// NETWORK 29
Ramp_Test_0(
    Enable := VCC_Ramp_Test_On,
    uExt := VCC_Ramp_Test_u_DCV_1,
    u0 := 0,
    uRetr := VCC_Ramp_Test_u_DCV_2,
    t0 := VCC_Test_t0,
    tRampUp := VCC_Ramp_Test_tR,
    tHold_Up := VCC_Ramp_Test_tHold_Up,
    tHold_Down := VCC_Ramp_Test_tHold_Down,
    tRampDown := VCC_Ramp_Test_tR,
    tWait := VCC_Ramp_Test_tWait,
    CyclicTime := UDP_Send.plcTime); // Ramp_Test
VCC_Anti_Dead_Band_v2_0(
    u_DCV_ref := Ramp_Test_0.Valve_Opening_Ref,
    DB_Up := VCC_Cntrl_DB_up,
    DB_Down := VCC_Cntrl_DB_down); // VCC_Anti_Dead_Band_v2
LREAL_TO_REAL(VCC_Anti_Dead_Band_v2_0.u_DCV);

// NETWORK 30
Ramp_Test_1(
    Enable := VCC_Ramp_Test_On,
    uExt := VCC_Ramp_Test_u_DCV_1,
    u0 := 0,
    uRetr := VCC_Ramp_Test_u_DCV_2,
    t0 := VCC_Test_t0,
    tRampUp := VCC_Ramp_Test_tR,
    tHold_Up := VCC_Ramp_Test_tHold_Up,
    tHold_Down := VCC_Ramp_Test_tHold_Down,
    tRampDown := VCC_Ramp_Test_tR,
    tWait := VCC_Ramp_Test_tWait,
    CyclicTime := UDP_Send.plcTime); // Ramp_Test
uRamp := LREAL_TO_REAL(Ramp_Test_1.Valve_Opening_Ref);

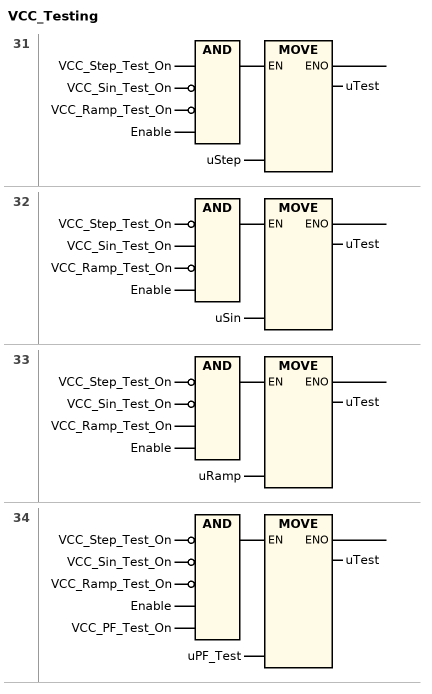
// NETWORK 31
IF VCC_Step_Test_On AND NOT VCC_Sin_Test_On AND NOT VCC_Ramp_Test_On AND Enable THEN uTest := uStep; END_IF

// NETWORK 32
IF NOT VCC_Step_Test_On AND VCC_Sin_Test_On AND NOT VCC_Ramp_Test_On AND Enable THEN uTest := uSin; END_IF

// NETWORK 33
IF NOT VCC_Step_Test_On AND NOT VCC_Sin_Test_On AND VCC_Ramp_Test_On AND Enable THEN uTest := uRamp; END_IF

// NETWORK 34
IF NOT VCC_Step_Test_On AND NOT VCC_Sin_Test_On AND NOT VCC_Ramp_Test_On AND Enable AND VCC_PF_Test_On THEN
    uTest := uPF_Test;
END_IF

END_PROGRAM

// IndraMotionMlc1/Application/VCC_StepFunction_Test
FUNCTION_BLOCK VCC_StepFunction_Test
VAR_INPUT
	Enable: BOOL;
	Extend_Opening_SP: LREAL;
	Neutral_Pos_SP: LREAL;
	Retract_Opening_SP: LREAL;
	CyclicTime: LREAL;
	t0: LREAL;
	t1: LREAL;
	t2: LREAL;
	t3: LREAL;
END_VAR
VAR_OUTPUT
	Valve_Opening_Ref: LREAL;
	EndTime: LREAL;
END_VAR
VAR
	tmp: LREAL;
	temp1: LREAL;
END_VAR


(* MATLAB Function: '<S1>/StepFunction' *)
(* MATLAB Function 'VCC_StepFunction_Test/StepFunction': '<S2>:1' *)
(* '<S2>:1:3' y = Neutral_Pos_SP; *)
(* '<S2>:1:5' if t>=0 &amp;&amp; t<t0 *)

IF (CyclicTime >= 0.0) AND (CyclicTime < t0) THEN 
    (* '<S2>:1:6' y = Neutral_Pos_SP; *)
    Valve_Opening_Ref := Neutral_Pos_SP;
ELSE 
    tmp := t0 + t1;

    IF (CyclicTime >= t0) AND (CyclicTime < tmp) THEN 
        (* '<S2>:1:7' elseif t>=(t0) &amp;&amp; t<(t0+t1) *)
        (* '<S2>:1:8' y = Extend_Opening_SP; *)
        Valve_Opening_Ref := Extend_Opening_SP;
    ELSE 
        temp1 := tmp + t2;

        IF (CyclicTime >= tmp) AND (CyclicTime < temp1) THEN 
            (* '<S2>:1:9' elseif t>=(t0+t1) &amp;&amp; t<(t0+t1+t2) *)
            (* '<S2>:1:10' y = Neutral_Pos_SP; *)
            Valve_Opening_Ref := Neutral_Pos_SP;
        ELSIF (CyclicTime >= temp1) AND (CyclicTime < (temp1 + t3)) THEN 
            (* '<S2>:1:11' elseif t>=(t0+t1+t2) &amp;&amp; t<(t0+t1+t2+t3) *)
            (* '<S2>:1:12' y = Retract_Opening_SP; *)
            Valve_Opening_Ref := Retract_Opening_SP;
        ELSE 
            (* '<S2>:1:13' else *)
            (* '<S2>:1:14' y = Neutral_Pos_SP; *)
            Valve_Opening_Ref := Neutral_Pos_SP;
        END_IF;

    END_IF;

END_IF;

(* Switch: '<S1>/Switch' *)
(* '<S2>:1:17' T = t0+t1+t2+t3; *)

IF  NOT Enable THEN 
    (* Outport: '<Root>/Valve_Opening_Ref' *)
    Valve_Opening_Ref := Neutral_Pos_SP;
END_IF;

(* End of Switch: '<S1>/Switch' *)


(* Outport: '<Root>/EndTime' incorporates:
 *  MATLAB Function: '<S1>/StepFunction' *)
EndTime := ((t0 + t1) + t2) + t3;

END_FUNCTION_BLOCK

// IndraMotionMlc1/Application/PF1
FUNCTION_BLOCK PF1
VAR_INPUT
	ssMethodType: SINT;
	Enable: BOOL;
	usDelay: LREAL;
	kQf: LREAL;
	HPF_Num1: LREAL;
	HPF_Num2: LREAL;
	HPF_Den1: LREAL;
	HPF_Den2: LREAL;
	pAsimbar: LREAL;
	pBsimbar: LREAL;
END_VAR
VAR_OUTPUT
	uPF: LREAL;
END_VAR
VAR
	HP_Filter_tmp: LREAL;
	VectorConcatenate: ARRAY[0..1] OF LREAL;
	VectorConcatenate1: ARRAY[0..1] OF LREAL;
	HP_Filter_states: LREAL;
END_VAR



CASE ssMethodType OF
    0: 
        (* InitializeConditions for DiscreteTransferFcn: '<S1>/HP_Filter' *)
        HP_Filter_states := 0.0;
    1: 
        (* SignalConversion: '<S1>/ConcatBufferAtVector ConcatenateIn1' *)
        VectorConcatenate[0] := HPF_Num1;
        (* SignalConversion: '<S1>/ConcatBufferAtVector ConcatenateIn2' *)
        VectorConcatenate[1] := HPF_Num2;
        (* SignalConversion: '<S1>/ConcatBufferAtVector Concatenate1In1' *)
        VectorConcatenate1[0] := HPF_Den1;
        (* SignalConversion: '<S1>/ConcatBufferAtVector Concatenate1In2' *)
        VectorConcatenate1[1] := HPF_Den2;
        (* DiscreteTransferFcn: '<S1>/HP_Filter' incorporates:
         *  Gain: '<S1>/Gain'
         *  Gain: '<S1>/Gain3'
         *  Gain: '<S1>/muC'
         *  Sum: '<S1>/Add' *)
        HP_Filter_tmp := (((100000.0 * pAsimbar) * 1.4083) - (100000.0 * pBsimbar)) - (VectorConcatenate1[1] * HP_Filter_states);
        (* Switch: '<S1>/Switch2' incorporates:
         *  Constant: '<S1>/Constant' *)

        IF Enable THEN 
            (* Switch: '<S1>/Switch1' incorporates:
             *  Constant: '<S1>/Constant'
             *  DiscreteTransferFcn: '<S1>/HP_Filter'
             *  Product: '<S1>/Product' *)

            IF usDelay > 2.0 THEN 
                uPF := ((VectorConcatenate[0] * HP_Filter_tmp) + (VectorConcatenate[1] * HP_Filter_states)) * kQf;
            ELSE 
                uPF := 0.0;
            END_IF;

            (* End of Switch: '<S1>/Switch1' *)
        ELSE 
            uPF := 0.0;
        END_IF;

        (* End of Switch: '<S1>/Switch2' *)
        

        (* Saturate: '<S1>/Saturation5' *)

        IF uPF >= 1.0 THEN 
            uPF := 1.0;
        ELSIF uPF <= -1.0 THEN 
            uPF := -1.0;
        END_IF;

        (* End of Saturate: '<S1>/Saturation5' *)
        

        (* Update for DiscreteTransferFcn: '<S1>/HP_Filter' *)
        HP_Filter_states := HP_Filter_tmp;
END_CASE;

END_FUNCTION_BLOCK

// IndraMotionMlc1/Application/PF2
FUNCTION_BLOCK PF2
VAR_INPUT
	ssMethodType: SINT;
	Enable: BOOL;
	usDelay: LREAL;
	kQf: LREAL;
	HPF_Num1: LREAL;
	HPF_Num2: LREAL;
	HPF_Den1: LREAL;
	HPF_Den2: LREAL;
	GVI_Num1: LREAL;
	GVI_Num2: LREAL;
	GVI_Num3: LREAL;
	GVI_Den1: LREAL;
	GVI_Den2: LREAL;
	GVI_Den3: LREAL;
	pAsimbar: LREAL;
	pBsimbar: LREAL;
END_VAR
VAR_OUTPUT
	uPF: LREAL;
END_VAR
VAR
	rtb_Add: LREAL;
	HP_Filter_tmp: LREAL;
	VectorConcatenate: ARRAY[0..1] OF LREAL;
	VectorConcatenate1: ARRAY[0..1] OF LREAL;
	VectorConcatenate2: ARRAY[0..2] OF LREAL;
	VectorConcatenate3: ARRAY[0..2] OF LREAL;
	HP_Filter_states: LREAL;
	Gv_Inv_states: ARRAY[0..1] OF LREAL;
END_VAR



CASE ssMethodType OF
    0: 
        (* InitializeConditions for DiscreteTransferFcn: '<S1>/HP_Filter' *)
        HP_Filter_states := 0.0;
        (* InitializeConditions for DiscreteTransferFcn: '<S1>/Gv_Inv' *)
        Gv_Inv_states[0] := 0.0;
        Gv_Inv_states[1] := 0.0;
    1: 
        (* SignalConversion: '<S1>/ConcatBufferAtVector ConcatenateIn1' *)
        VectorConcatenate[0] := HPF_Num1;
        (* SignalConversion: '<S1>/ConcatBufferAtVector ConcatenateIn2' *)
        VectorConcatenate[1] := HPF_Num2;
        (* SignalConversion: '<S1>/ConcatBufferAtVector Concatenate1In1' *)
        VectorConcatenate1[0] := HPF_Den1;
        (* SignalConversion: '<S1>/ConcatBufferAtVector Concatenate1In2' *)
        VectorConcatenate1[1] := HPF_Den2;
        (* DiscreteTransferFcn: '<S1>/HP_Filter' incorporates:
         *  Gain: '<S1>/Gain'
         *  Gain: '<S1>/Gain3'
         *  Gain: '<S1>/muC'
         *  Sum: '<S1>/Add' *)
        HP_Filter_tmp := (((100000.0 * pAsimbar) * 1.4083) - (100000.0 * pBsimbar)) - (VectorConcatenate1[1] * HP_Filter_states);
        (* SignalConversion: '<S1>/ConcatBufferAtVector Concatenate2In1' *)
        VectorConcatenate2[0] := GVI_Num1;
        (* SignalConversion: '<S1>/ConcatBufferAtVector Concatenate2In2' *)
        VectorConcatenate2[1] := GVI_Num2;
        (* SignalConversion: '<S1>/ConcatBufferAtVector Concatenate2In3' *)
        VectorConcatenate2[2] := GVI_Num3;
        (* SignalConversion: '<S1>/ConcatBufferAtVector Concatenate3In1' *)
        VectorConcatenate3[0] := GVI_Den1;
        (* SignalConversion: '<S1>/ConcatBufferAtVector Concatenate3In2' *)
        VectorConcatenate3[1] := GVI_Den2;
        (* SignalConversion: '<S1>/ConcatBufferAtVector Concatenate3In3' *)
        VectorConcatenate3[2] := GVI_Den3;
        (* DiscreteTransferFcn: '<S1>/Gv_Inv' incorporates:
         *  DiscreteTransferFcn: '<S1>/HP_Filter'
         *  Product: '<S1>/Product' *)
        rtb_Add := ((((VectorConcatenate[0] * HP_Filter_tmp) + (VectorConcatenate[1] * HP_Filter_states)) * kQf) - (VectorConcatenate3[1] * Gv_Inv_states[0])) - (VectorConcatenate3[2] * Gv_Inv_states[1]);
        (* Switch: '<S1>/Switch2' incorporates:
         *  Constant: '<S1>/Constant' *)

        IF Enable THEN 
            (* Switch: '<S1>/Switch1' incorporates:
             *  Constant: '<S1>/Constant'
             *  DiscreteTransferFcn: '<S1>/Gv_Inv' *)

            IF usDelay > 2.0 THEN 
                uPF := ((VectorConcatenate2[0] * rtb_Add) + (VectorConcatenate2[1] * Gv_Inv_states[0])) + (VectorConcatenate2[2] * Gv_Inv_states[1]);
            ELSE 
                uPF := 0.0;
            END_IF;

            (* End of Switch: '<S1>/Switch1' *)
        ELSE 
            uPF := 0.0;
        END_IF;

        (* End of Switch: '<S1>/Switch2' *)
        

        (* Saturate: '<S1>/Saturation5' *)

        IF uPF >= 1.0 THEN 
            uPF := 1.0;
        ELSIF uPF <= -1.0 THEN 
            uPF := -1.0;
        END_IF;

        (* End of Saturate: '<S1>/Saturation5' *)
        

        (* Update for DiscreteTransferFcn: '<S1>/HP_Filter' *)
        HP_Filter_states := HP_Filter_tmp;
        (* Update for DiscreteTransferFcn: '<S1>/Gv_Inv' *)
        Gv_Inv_states[1] := Gv_Inv_states[0];
        Gv_Inv_states[0] := rtb_Add;
END_CASE;

END_FUNCTION_BLOCK

// IndraMotionMlc1/Application/HPPF_pB
FUNCTION_BLOCK HPPF_pB
VAR_INPUT
	ssMethodType: SINT;
	Enable: BOOL;
	usDelay: LREAL;
	kQf: LREAL;
	HPF_Num1: LREAL;
	HPF_Num2: LREAL;
	HPF_Den1: LREAL;
	HPF_Den2: LREAL;
	pBsimbar: LREAL;
END_VAR
VAR_OUTPUT
	uPF: LREAL;
END_VAR
VAR
	HP_Filter_tmp: LREAL;
	VectorConcatenate: ARRAY[0..1] OF LREAL;
	VectorConcatenate1: ARRAY[0..1] OF LREAL;
	HP_Filter_states: LREAL;
END_VAR



CASE ssMethodType OF
    0: 
        (* InitializeConditions for DiscreteTransferFcn: '<S1>/HP_Filter' *)
        HP_Filter_states := 0.0;
    1: 
        (* SignalConversion: '<S1>/ConcatBufferAtVector ConcatenateIn1' *)
        VectorConcatenate[0] := HPF_Num1;
        (* SignalConversion: '<S1>/ConcatBufferAtVector ConcatenateIn2' *)
        VectorConcatenate[1] := HPF_Num2;
        (* SignalConversion: '<S1>/ConcatBufferAtVector Concatenate1In1' *)
        VectorConcatenate1[0] := HPF_Den1;
        (* SignalConversion: '<S1>/ConcatBufferAtVector Concatenate1In2' *)
        VectorConcatenate1[1] := HPF_Den2;
        (* DiscreteTransferFcn: '<S1>/HP_Filter' incorporates:
         *  Gain: '<S1>/Gain3' *)
        HP_Filter_tmp := (100000.0 * pBsimbar) - (VectorConcatenate1[1] * HP_Filter_states);
        (* Switch: '<S1>/Switch2' incorporates:
         *  Constant: '<S1>/Constant' *)

        IF Enable THEN 
            (* Switch: '<S1>/Switch1' incorporates:
             *  Constant: '<S1>/Constant'
             *  DiscreteTransferFcn: '<S1>/HP_Filter'
             *  Product: '<S1>/Product' *)

            IF usDelay > 2.0 THEN 
                uPF := ((VectorConcatenate[0] * HP_Filter_tmp) + (VectorConcatenate[1] * HP_Filter_states)) * kQf;
            ELSE 
                uPF := 0.0;
            END_IF;

            (* End of Switch: '<S1>/Switch1' *)
        ELSE 
            uPF := 0.0;
        END_IF;

        (* End of Switch: '<S1>/Switch2' *)
        

        (* Saturate: '<S1>/Saturation5' *)

        IF uPF >= 1.0 THEN 
            uPF := 1.0;
        ELSIF uPF <= -1.0 THEN 
            uPF := -1.0;
        END_IF;

        (* End of Saturate: '<S1>/Saturation5' *)
        

        (* Update for DiscreteTransferFcn: '<S1>/HP_Filter' *)
        HP_Filter_states := HP_Filter_tmp;
END_CASE;

END_FUNCTION_BLOCK

// IndraMotionMlc1/Application/HPPF2_pB
FUNCTION_BLOCK HPPF2_pB
VAR_INPUT
	ssMethodType: SINT;
	Enable: BOOL;
	usDelay: LREAL;
	kQf: LREAL;
	HPF_Num1: LREAL;
	HPF_Num2: LREAL;
	HPF_Den1: LREAL;
	HPF_Den2: LREAL;
	GVI_Num1: LREAL;
	GVI_Num2: LREAL;
	GVI_Num3: LREAL;
	GVI_Den1: LREAL;
	GVI_Den2: LREAL;
	GVI_Den3: LREAL;
	pBsimbar: LREAL;
END_VAR
VAR_OUTPUT
	uPF: LREAL;
END_VAR
VAR
	rtb_Gain3: LREAL;
	HP_Filter_tmp: LREAL;
	VectorConcatenate: ARRAY[0..1] OF LREAL;
	VectorConcatenate1: ARRAY[0..1] OF LREAL;
	VectorConcatenate2: ARRAY[0..2] OF LREAL;
	VectorConcatenate3: ARRAY[0..2] OF LREAL;
	HP_Filter_states: LREAL;
	Gv_Inv_states: ARRAY[0..1] OF LREAL;
END_VAR



CASE ssMethodType OF
    0: 
        (* InitializeConditions for DiscreteTransferFcn: '<S1>/HP_Filter' *)
        HP_Filter_states := 0.0;
        (* InitializeConditions for DiscreteTransferFcn: '<S1>/Gv_Inv' *)
        Gv_Inv_states[0] := 0.0;
        Gv_Inv_states[1] := 0.0;
    1: 
        (* SignalConversion: '<S1>/ConcatBufferAtVector ConcatenateIn1' *)
        VectorConcatenate[0] := HPF_Num1;
        (* SignalConversion: '<S1>/ConcatBufferAtVector ConcatenateIn2' *)
        VectorConcatenate[1] := HPF_Num2;
        (* SignalConversion: '<S1>/ConcatBufferAtVector Concatenate1In1' *)
        VectorConcatenate1[0] := HPF_Den1;
        (* SignalConversion: '<S1>/ConcatBufferAtVector Concatenate1In2' *)
        VectorConcatenate1[1] := HPF_Den2;
        (* DiscreteTransferFcn: '<S1>/HP_Filter' incorporates:
         *  Gain: '<S1>/Gain3' *)
        HP_Filter_tmp := (100000.0 * pBsimbar) - (VectorConcatenate1[1] * HP_Filter_states);
        (* SignalConversion: '<S1>/ConcatBufferAtVector Concatenate2In1' *)
        VectorConcatenate2[0] := GVI_Num1;
        (* SignalConversion: '<S1>/ConcatBufferAtVector Concatenate2In2' *)
        VectorConcatenate2[1] := GVI_Num2;
        (* SignalConversion: '<S1>/ConcatBufferAtVector Concatenate2In3' *)
        VectorConcatenate2[2] := GVI_Num3;
        (* SignalConversion: '<S1>/ConcatBufferAtVector Concatenate3In1' *)
        VectorConcatenate3[0] := GVI_Den1;
        (* SignalConversion: '<S1>/ConcatBufferAtVector Concatenate3In2' *)
        VectorConcatenate3[1] := GVI_Den2;
        (* SignalConversion: '<S1>/ConcatBufferAtVector Concatenate3In3' *)
        VectorConcatenate3[2] := GVI_Den3;
        (* DiscreteTransferFcn: '<S1>/Gv_Inv' incorporates:
         *  DiscreteTransferFcn: '<S1>/HP_Filter'
         *  Product: '<S1>/Product' *)
        rtb_Gain3 := ((((VectorConcatenate[0] * HP_Filter_tmp) + (VectorConcatenate[1] * HP_Filter_states)) * kQf) - (VectorConcatenate3[1] * Gv_Inv_states[0])) - (VectorConcatenate3[2] * Gv_Inv_states[1]);
        (* Switch: '<S1>/Switch2' incorporates:
         *  Constant: '<S1>/Constant' *)

        IF Enable THEN 
            (* Switch: '<S1>/Switch1' incorporates:
             *  Constant: '<S1>/Constant'
             *  DiscreteTransferFcn: '<S1>/Gv_Inv' *)

            IF usDelay > 2.0 THEN 
                uPF := ((VectorConcatenate2[0] * rtb_Gain3) + (VectorConcatenate2[1] * Gv_Inv_states[0])) + (VectorConcatenate2[2] * Gv_Inv_states[1]);
            ELSE 
                uPF := 0.0;
            END_IF;

            (* End of Switch: '<S1>/Switch1' *)
        ELSE 
            uPF := 0.0;
        END_IF;

        (* End of Switch: '<S1>/Switch2' *)
        

        (* Saturate: '<S1>/Saturation5' *)

        IF uPF >= 1.0 THEN 
            uPF := 1.0;
        ELSIF uPF <= -1.0 THEN 
            uPF := -1.0;
        END_IF;

        (* End of Saturate: '<S1>/Saturation5' *)
        

        (* Update for DiscreteTransferFcn: '<S1>/HP_Filter' *)
        HP_Filter_states := HP_Filter_tmp;
        (* Update for DiscreteTransferFcn: '<S1>/Gv_Inv' *)
        Gv_Inv_states[1] := Gv_Inv_states[0];
        Gv_Inv_states[0] := rtb_Gain3;
END_CASE;

END_FUNCTION_BLOCK

// IndraMotionMlc1/Application/HPPF_pA
FUNCTION_BLOCK HPPF_pA
VAR_INPUT
	ssMethodType: SINT;
	Enable: BOOL;
	usDelay: LREAL;
	kQf: LREAL;
	HPF_Num1: LREAL;
	HPF_Num2: LREAL;
	HPF_Den1: LREAL;
	HPF_Den2: LREAL;
	pAsimbar: LREAL;
END_VAR
VAR_OUTPUT
	uPF: LREAL;
END_VAR
VAR
	HP_Filter_tmp: LREAL;
	VectorConcatenate: ARRAY[0..1] OF LREAL;
	VectorConcatenate1: ARRAY[0..1] OF LREAL;
	HP_Filter_states: LREAL;
END_VAR



CASE ssMethodType OF
    0: 
        (* InitializeConditions for DiscreteTransferFcn: '<S1>/HP_Filter' *)
        HP_Filter_states := 0.0;
    1: 
        (* SignalConversion: '<S1>/ConcatBufferAtVector ConcatenateIn1' *)
        VectorConcatenate[0] := HPF_Num1;
        (* SignalConversion: '<S1>/ConcatBufferAtVector ConcatenateIn2' *)
        VectorConcatenate[1] := HPF_Num2;
        (* SignalConversion: '<S1>/ConcatBufferAtVector Concatenate1In1' *)
        VectorConcatenate1[0] := HPF_Den1;
        (* SignalConversion: '<S1>/ConcatBufferAtVector Concatenate1In2' *)
        VectorConcatenate1[1] := HPF_Den2;
        (* DiscreteTransferFcn: '<S1>/HP_Filter' incorporates:
         *  Gain: '<S1>/Gain' *)
        HP_Filter_tmp := (100000.0 * pAsimbar) - (VectorConcatenate1[1] * HP_Filter_states);
        (* Switch: '<S1>/Switch2' incorporates:
         *  Constant: '<S1>/Constant' *)

        IF Enable THEN 
            (* Switch: '<S1>/Switch1' incorporates:
             *  Constant: '<S1>/Constant'
             *  DiscreteTransferFcn: '<S1>/HP_Filter'
             *  Product: '<S1>/Product' *)

            IF usDelay > 2.0 THEN 
                uPF := ((VectorConcatenate[0] * HP_Filter_tmp) + (VectorConcatenate[1] * HP_Filter_states)) * kQf;
            ELSE 
                uPF := 0.0;
            END_IF;

            (* End of Switch: '<S1>/Switch1' *)
        ELSE 
            uPF := 0.0;
        END_IF;

        (* End of Switch: '<S1>/Switch2' *)
        

        (* Saturate: '<S1>/Saturation5' *)

        IF uPF >= 1.0 THEN 
            uPF := 1.0;
        ELSIF uPF <= -1.0 THEN 
            uPF := -1.0;
        END_IF;

        (* End of Saturate: '<S1>/Saturation5' *)
        

        (* Update for DiscreteTransferFcn: '<S1>/HP_Filter' *)
        HP_Filter_states := HP_Filter_tmp;
END_CASE;

END_FUNCTION_BLOCK

// IndraMotionMlc1/Application/HPPF2_pA
FUNCTION_BLOCK HPPF2_pA
VAR_INPUT
	ssMethodType: SINT;
	Enable: BOOL;
	usDelay: LREAL;
	kQf: LREAL;
	HPF_Num1: LREAL;
	HPF_Num2: LREAL;
	HPF_Den1: LREAL;
	HPF_Den2: LREAL;
	GVI_Num1: LREAL;
	GVI_Num2: LREAL;
	GVI_Num3: LREAL;
	GVI_Den1: LREAL;
	GVI_Den2: LREAL;
	GVI_Den3: LREAL;
	pAsimbar: LREAL;
END_VAR
VAR_OUTPUT
	uPF: LREAL;
END_VAR
VAR
	rtb_Gain: LREAL;
	HP_Filter_tmp: LREAL;
	VectorConcatenate: ARRAY[0..1] OF LREAL;
	VectorConcatenate1: ARRAY[0..1] OF LREAL;
	VectorConcatenate2: ARRAY[0..2] OF LREAL;
	VectorConcatenate3: ARRAY[0..2] OF LREAL;
	HP_Filter_states: LREAL;
	Gv_Inv_states: ARRAY[0..1] OF LREAL;
END_VAR



CASE ssMethodType OF
    0: 
        (* InitializeConditions for DiscreteTransferFcn: '<S1>/HP_Filter' *)
        HP_Filter_states := 0.0;
        (* InitializeConditions for DiscreteTransferFcn: '<S1>/Gv_Inv' *)
        Gv_Inv_states[0] := 0.0;
        Gv_Inv_states[1] := 0.0;
    1: 
        (* SignalConversion: '<S1>/ConcatBufferAtVector ConcatenateIn1' *)
        VectorConcatenate[0] := HPF_Num1;
        (* SignalConversion: '<S1>/ConcatBufferAtVector ConcatenateIn2' *)
        VectorConcatenate[1] := HPF_Num2;
        (* SignalConversion: '<S1>/ConcatBufferAtVector Concatenate1In1' *)
        VectorConcatenate1[0] := HPF_Den1;
        (* SignalConversion: '<S1>/ConcatBufferAtVector Concatenate1In2' *)
        VectorConcatenate1[1] := HPF_Den2;
        (* DiscreteTransferFcn: '<S1>/HP_Filter' incorporates:
         *  Gain: '<S1>/Gain' *)
        HP_Filter_tmp := (100000.0 * pAsimbar) - (VectorConcatenate1[1] * HP_Filter_states);
        (* SignalConversion: '<S1>/ConcatBufferAtVector Concatenate2In1' *)
        VectorConcatenate2[0] := GVI_Num1;
        (* SignalConversion: '<S1>/ConcatBufferAtVector Concatenate2In2' *)
        VectorConcatenate2[1] := GVI_Num2;
        (* SignalConversion: '<S1>/ConcatBufferAtVector Concatenate2In3' *)
        VectorConcatenate2[2] := GVI_Num3;
        (* SignalConversion: '<S1>/ConcatBufferAtVector Concatenate3In1' *)
        VectorConcatenate3[0] := GVI_Den1;
        (* SignalConversion: '<S1>/ConcatBufferAtVector Concatenate3In2' *)
        VectorConcatenate3[1] := GVI_Den2;
        (* SignalConversion: '<S1>/ConcatBufferAtVector Concatenate3In3' *)
        VectorConcatenate3[2] := GVI_Den3;
        (* DiscreteTransferFcn: '<S1>/Gv_Inv' incorporates:
         *  DiscreteTransferFcn: '<S1>/HP_Filter'
         *  Product: '<S1>/Product' *)
        rtb_Gain := ((((VectorConcatenate[0] * HP_Filter_tmp) + (VectorConcatenate[1] * HP_Filter_states)) * kQf) - (VectorConcatenate3[1] * Gv_Inv_states[0])) - (VectorConcatenate3[2] * Gv_Inv_states[1]);
        (* Switch: '<S1>/Switch2' incorporates:
         *  Constant: '<S1>/Constant' *)

        IF Enable THEN 
            (* Switch: '<S1>/Switch1' incorporates:
             *  Constant: '<S1>/Constant'
             *  DiscreteTransferFcn: '<S1>/Gv_Inv' *)

            IF usDelay > 2.0 THEN 
                uPF := ((VectorConcatenate2[0] * rtb_Gain) + (VectorConcatenate2[1] * Gv_Inv_states[0])) + (VectorConcatenate2[2] * Gv_Inv_states[1]);
            ELSE 
                uPF := 0.0;
            END_IF;

            (* End of Switch: '<S1>/Switch1' *)
        ELSE 
            uPF := 0.0;
        END_IF;

        (* End of Switch: '<S1>/Switch2' *)
        

        (* Saturate: '<S1>/Saturation5' *)

        IF uPF >= 1.0 THEN 
            uPF := 1.0;
        ELSIF uPF <= -1.0 THEN 
            uPF := -1.0;
        END_IF;

        (* End of Saturate: '<S1>/Saturation5' *)
        

        (* Update for DiscreteTransferFcn: '<S1>/HP_Filter' *)
        HP_Filter_states := HP_Filter_tmp;
        (* Update for DiscreteTransferFcn: '<S1>/Gv_Inv' *)
        Gv_Inv_states[1] := Gv_Inv_states[0];
        Gv_Inv_states[0] := rtb_Gain;
END_CASE;

END_FUNCTION_BLOCK

// IndraMotionMlc1/Application/VCC_Anti_Dead_Band_v2
FUNCTION_BLOCK VCC_Anti_Dead_Band_v2
VAR_INPUT
	u_DCV_ref: LREAL;
	DB_Up: LREAL;
	DB_Down: LREAL;
END_VAR
VAR_OUTPUT
	u_DCV: LREAL;
END_VAR
VAR
END_VAR


(* MATLAB Function: '<S1>/Anti_Dead_Band' *)
(* MATLAB Function 'Anti_Dead_Band/Anti_Dead_Band': '<S2>:1' *)
(* '<S2>:1:3' u_DCV = 0; *)
(* '<S2>:1:5' if u_DCV_ref < -0.001 *)

        IF u_DCV_ref < -0.001 THEN 
            (* Outport: '<Root>/u_DCV' *)
            (* '<S2>:1:9' elseif (u_DCV_ref < -0.001) *)
            (* '<S2>:1:10' u_DCV = -DB_Up + (1-DB_Up)*u_DCV_ref; *)
            u_DCV := ((1.0 - DB_Up) * u_DCV_ref) + ( -DB_Up);
        ELSIF u_DCV_ref > 0.001 THEN 
            (* Outport: '<Root>/u_DCV' *)
            (* '<S2>:1:11' elseif (u_DCV_ref > 0.001) *)
            (* '<S2>:1:12' u_DCV = DB_Down + (1-DB_Down)*u_DCV_ref; *)
            u_DCV := ((1.0 - DB_Down) * u_DCV_ref) + DB_Down;
        ELSE 
            (* Outport: '<Root>/u_DCV' *)
            (* '<S2>:1:13' else *)
            (* '<S2>:1:14' u_DCV = 0; *)
            u_DCV := 0.0;
        END_IF;

(* End of MATLAB Function: '<S1>/Anti_Dead_Band' *)

END_FUNCTION_BLOCK

// IndraMotionMlc1/Application/VCC_StepFunction
FUNCTION_BLOCK VCC_StepFunction
VAR_INPUT
	Enable: BOOL;
	u_SP: LREAL;
	CyclicTime: LREAL;
	t0: LREAL;
	t1: LREAL;
END_VAR
VAR_OUTPUT
	u_ref: LREAL;
	EndTime: LREAL;
END_VAR
VAR
END_VAR


(* MATLAB Function: '<S1>/StepFunction' *)
(* MATLAB Function 'VCC_StepFunction/StepFunction': '<S2>:1' *)
(* '<S2>:1:3' y = 0; *)
(* '<S2>:1:5' if t>=0 &amp;&amp; t<t0 *)

IF (CyclicTime >= 0.0) AND (CyclicTime < t0) THEN 
    (* '<S2>:1:6' y = 0; *)
    u_ref := 0.0;
ELSIF (CyclicTime >= t0) AND (CyclicTime < (t0 + t1)) THEN 
    (* '<S2>:1:7' elseif t>=(t0) &amp;&amp; t<(t0+t1) *)
    (* '<S2>:1:8' y = u_SP; *)
    u_ref := u_SP;
ELSE 
    (* '<S2>:1:9' else *)
    (* '<S2>:1:10' y = 0; *)
    u_ref := 0.0;
END_IF;

(* Switch: '<S1>/Switch' *)
(* '<S2>:1:13' T = t0+t1; *)

IF  NOT Enable THEN 
    (* Outport: '<Root>/u_ref' incorporates:
     *  Constant: '<S1>/Constant' *)
    u_ref := 0.0;
END_IF;

(* End of Switch: '<S1>/Switch' *)


(* Outport: '<Root>/EndTime' incorporates:
 *  MATLAB Function: '<S1>/StepFunction' *)
EndTime := t0 + t1;

END_FUNCTION_BLOCK

// IndraMotionMlc1/Application/VCC_Step_Function_Validation
FUNCTION_BLOCK VCC_Step_Function_Validation
VAR_INPUT
	Enable: BOOL;
	u_SP: LREAL;
	uS0: LREAL;
	DB: LREAL;
	CyclicTime: LREAL;
	t0: LREAL;
	tHold1: LREAL;
	tStep: LREAL;
	tHold2: LREAL;
END_VAR
VAR_OUTPUT
	u_ref: LREAL;
	EndTime: LREAL;
END_VAR
VAR
	tmp: LREAL;
	temp1: LREAL;
END_VAR


(* MATLAB Function: '<S1>/StepFunction' *)
(* MATLAB Function 'VCC_Step_Function_Validation/StepFunction': '<S2>:1' *)
(* '<S2>:1:2' y = 0; *)
(* '<S2>:1:4' if t>=0 &amp;&amp; t<t0 *)

IF (CyclicTime >= 0.0) AND (CyclicTime < t0) THEN 
    (* '<S2>:1:5' y = (uS0+DB)/t0*t; *)
    u_ref := ((uS0 + DB) / t0) * CyclicTime;
ELSE 
    tmp := t0 + tHold1;

    IF (CyclicTime >= t0) AND (CyclicTime < tmp) THEN 
        (* '<S2>:1:6' elseif t>=(t0) &amp;&amp; t<(t0+t1) *)
        (* '<S2>:1:7' y = uS0+DB; *)
        u_ref := uS0 + DB;
    ELSE 
        temp1 := tmp + tStep;

        IF (CyclicTime >= tmp) AND (CyclicTime < temp1) THEN 
            (* '<S2>:1:8' elseif t>=(t0+t1) &amp;&amp; t<(t0+t1+t2) *)
            (* '<S2>:1:9' y = u_SP+DB; *)
            u_ref := u_SP + DB;
        ELSIF (CyclicTime >= temp1) AND (CyclicTime < (temp1 + tHold2)) THEN 
            (* '<S2>:1:10' elseif t>=(t0+t1+t2) &amp;&amp; t<(t0+t1+t2+t3) *)
            (* '<S2>:1:11' y = uS0+DB; *)
            u_ref := uS0 + DB;
        ELSE 
            (* '<S2>:1:12' else *)
            (* '<S2>:1:13' y = 0; *)
            u_ref := 0.0;
        END_IF;

    END_IF;

END_IF;

(* Switch: '<S1>/Switch' *)
(* '<S2>:1:16' T = t0+t1+t2+t3; *)

IF  NOT Enable THEN 
    (* Outport: '<Root>/u_ref' incorporates:
     *  Constant: '<S1>/Constant' *)
    u_ref := 0.0;
END_IF;

(* End of Switch: '<S1>/Switch' *)


(* Outport: '<Root>/EndTime' incorporates:
 *  MATLAB Function: '<S1>/StepFunction' *)
EndTime := ((t0 + tHold1) + tStep) + tHold2;

END_FUNCTION_BLOCK

// IndraMotionMlc1/Application/Ramp_Test
FUNCTION_BLOCK Ramp_Test
VAR_INPUT
	Enable: BOOL;
	uExt: LREAL;
	u0: LREAL;
	uRetr: LREAL;
	t0: LREAL;
	tRampUp: LREAL;
	tHold_Up: LREAL;
	tHold_Down: LREAL;
	tRampDown: LREAL;
	tWait: LREAL;
	CyclicTime: LREAL;
END_VAR
VAR_OUTPUT
	Valve_Opening_Ref: LREAL;
	T: LREAL;
END_VAR
VAR
	slopeExt: LREAL;
	slopeRetr: LREAL;
	tmp: LREAL;
	temp1: LREAL;
END_VAR


(* MATLAB Function: '<S1>/WaveSignal' *)
(* MATLAB Function 'Ramp_Test/WaveSignal': '<S2>:1' *)
(* '<S2>:1:2' slopeExt=u0-uExt; *)
slopeExt := u0 - uExt;
(* '<S2>:1:3' slopeRetr=uRetr-u0; *)
slopeRetr := uRetr - u0;
(* '<S2>:1:4' t1=tRampUp; *)
(* '<S2>:1:5' t2=tHold_Up; *)
(* '<S2>:1:6' t3=tRampDown; *)
(* '<S2>:1:7' t4=tWait; *)
(* '<S2>:1:8' t5=t1; *)
(* '<S2>:1:9' t6=t2; *)
(* '<S2>:1:10' t7=t3; *)
(* '<S2>:1:12' if t>=0 &amp;&amp; t<t0 *)

IF (CyclicTime >= 0.0) AND (CyclicTime < t0) THEN 
    (* '<S2>:1:13' u = u0; *)
    Valve_Opening_Ref := u0;
ELSE 
    tmp := t0 + tRampUp;

    IF (CyclicTime >= t0) AND (CyclicTime < tmp) THEN 
        (* '<S2>:1:14' elseif t>=t0 &amp;&amp; t<(t0+t1) *)
        (* '<S2>:1:15' u = u0-(slopeExt/t1)*(t-t0); *)
        Valve_Opening_Ref := u0 - ((slopeExt / tRampUp) * (CyclicTime - t0));
    ELSE 
        temp1 := tmp + tHold_Up;

        IF (CyclicTime >= tmp) AND (CyclicTime < temp1) THEN 
            (* '<S2>:1:16' elseif t>=(t0+t1) &amp;&amp; t<(t0+t1+t2) *)
            (* '<S2>:1:17' u = uExt; *)
            Valve_Opening_Ref := uExt;
        ELSE 
            tmp := temp1 + tRampDown;

            IF (CyclicTime >= temp1) AND (CyclicTime < tmp) THEN 
                (* '<S2>:1:18' elseif t>=(t0+t1+t2) &amp;&amp; t<(t0+t1+t2+t3) *)
                (* '<S2>:1:19' u = uExt+(slopeExt/t3)*(t-(t0+t1+t2)); *)
                Valve_Opening_Ref := ((CyclicTime - temp1) * (slopeExt / tRampDown)) + uExt;
            ELSE 
                temp1 := tmp + tWait;

                IF (CyclicTime >= tmp) AND (CyclicTime < temp1) THEN 
                    (* '<S2>:1:20' elseif t>=(t0+t1+t2+t3) &amp;&amp; t<(t0+t1+t2+t3+t4) *)
                    (* '<S2>:1:21' u = u0; *)
                    Valve_Opening_Ref := u0;
                ELSE 
                    tmp := temp1 + tRampUp;

                    IF (CyclicTime >= temp1) AND (CyclicTime < tmp) THEN 
                        (* '<S2>:1:22' elseif t>=(t0+t1+t2+t3+t4) &amp;&amp; t<(t0+t1+t2+t3+t4+t5) *)
                        (* '<S2>:1:23' u = u0+(slopeRetr/t5)*(t-(t0+t1+t2+t3+t4)); *)
                        Valve_Opening_Ref := ((CyclicTime - temp1) * (slopeRetr / tRampUp)) + u0;
                    ELSE 
                        temp1 := tmp + tHold_Down;

                        IF (CyclicTime >= tmp) AND (CyclicTime < temp1) THEN 
                            (* '<S2>:1:24' elseif t>=(t0+t1+t2+t3+t4+t5) &amp;&amp; t<(t0+t1+t2+t3+t4+t5+t6) *)
                            (* '<S2>:1:25' u = uRetr; *)
                            Valve_Opening_Ref := uRetr;
                        ELSIF (CyclicTime >= temp1) AND (CyclicTime < (temp1 + tRampDown)) THEN 
                            (* '<S2>:1:26' elseif t>=(t0+t1+t2+t3+t4+t5+t6) &amp;&amp; t<(t0+t1+t2+t3+t4+t5+t6+t7) *)
                            (* '<S2>:1:27' u = uRetr-(slopeRetr/t3)*(t-(t0+t1+t2+t3+t4+t5+t6)); *)
                            Valve_Opening_Ref := uRetr - ((CyclicTime - temp1) * (slopeRetr / tRampDown));
                        ELSE 
                            (* '<S2>:1:28' else *)
                            (* '<S2>:1:29' u = u0; *)
                            Valve_Opening_Ref := u0;
                        END_IF;

                    END_IF;

                END_IF;

            END_IF;

        END_IF;

    END_IF;

END_IF;

(* Switch: '<S1>/Switch' *)
(* '<S2>:1:32' T = t0+t1+t2+t3+t4+t5+t6+t7; *)

IF  NOT Enable THEN 
    (* Outport: '<Root>/Valve_Opening_Ref' *)
    Valve_Opening_Ref := u0;
END_IF;

(* End of Switch: '<S1>/Switch' *)


(* Outport: '<Root>/T' incorporates:
 *  MATLAB Function: '<S1>/WaveSignal' *)
T := ((((((t0 + tRampUp) + tHold_Up) + tRampDown) + tWait) + tRampUp) + tHold_Down) + tRampDown;

END_FUNCTION_BLOCK

// IndraMotionMlc1/Application/VCC_Controller
PROGRAM VCC_Controller
VAR_INPUT
	 Enable: BOOL;
END_VAR
VAR_OUTPUT
	u_Closed_Loop: REAL;
END_VAR
VAR
	VCC_PI_Controller_0: VCC_PI_Controller;
	kFF: LREAL;
	MaxError: LREAL := 1;
	MinError: LREAL := -1;
	uFB: LREAL;
	uFF: LREAL;
	ErrorSignal: LREAL;
	ZeroSignal: LREAL := 0.00;
    Reset_Integrator: LREAL;
    VCC_Joystick_vel_ref_0: VCC_Joystick_vel_ref;
	Vel_Ref_Manual: LREAL;
	Pos_Ref_Gen: LREAL;
	Vel_Ref: LREAL;
    Pos_Ref: LREAL;
	test: LREAL;
	AutoPLCtime_start: LREAL;
	SPtime: LREAL;
	SPtimereset: LREAL; 
	u_Manual_FeedForward: LREAL;
	Vel_Ref_Joystick: LREAL;
	kFF_Manual: LREAL;
    u_Manual_FF: LREAL;
	uCTRL: LREAL;	
	VCC_Anti_Dead_Band_v2_0: VCC_Anti_Dead_Band_v2;
	uDCV_ref: REAL;
	uDCV: LREAL;
	SP_Gen_Vel_Ref: LREAL;
	u_CTRL: LREAL;
	VCC_Anti_Dead_Band_v2_1: VCC_Anti_Dead_Band_v2;
	VCC_Controller_FF_PI_AD_v05_0: VCC_Controller_FF_PI_AD_v05;
	VCC_Controller_FF_PI_AD_0: VCC_Controller_FF_PI_AD;
	u_FF: LREAL;
	u_P_cntr: LREAL;
	u_I_cntr: LREAL;
	k_P: LREAL;
	VCC_SP_Ramp_Generator_0: VCC_SP_Ramp_Generator;
	Ramp_Pos_Ref_Gen: LREAL;
	Ramp_Vel_Ref_Gen: LREAL;
	S_shape_Pos_Ref_Gen: LREAL;
	S_shape_Vel_Ref_Gen: LREAL;
	S_shape_Profile_0: S_shape_Profile;
	Ramp_Profile_0: Ramp_Profile;
	Motion_Reset_Time: LREAL;
	T_Ramp: LREAL;
	T_S_shape: LREAL;
	VCC_Controller_PI_FF_0: VCC_Controller_PI_FF;
	uPF1: LREAL;
	uPF2: LREAL;
	uPF11: LREAL;
	uPF_Test_DB: REAL;
	uPF_Joy: REAL;
	uJoy: REAL;
	uLPPF: LREAL;
	uStep_ref: LREAL;
	HPPF_pB_0: HPPF_pB;
	uPF_pB: LREAL;
	HPPF2_pB_0: HPPF2_pB;
	uPF_pB_vInfOFF: LREAL;
	uPF_pB_vInfOn: LREAL;
	uPF_pL: LREAL;
	HPPF_pA_0: HPPF_pA;
	uPF_pA: LREAL;
	HPPF2_pA_0: HPPF2_pA;
	uPF_pA_vInfOn: LREAL;
	uPF_pA_vInfOff: LREAL;
		DB: LREAL;
	uPF: LREAL;
	PF2_0: PF2;
	JoyStick_VCC_0: JoyStick_VCC;
	uPF_Test: REAL;
	PF1_0: PF1;
	VCC_Controller_PFB_0: VCC_Controller_PFB;
	VCC_VFF_0: VCC_VFF;
	VCC_Cntrl_Error: LREAL;
	SR_0: SR;
	FBC_Enable: BOOL;
	R_TRIG_0: R_TRIG;
	R_TRIG_1: R_TRIG;
	VCC_StepFunction_0: VCC_StepFunction;
	Step_Pos_Ref: LREAL;
	VCC_Pos_Step_0: VCC_Pos_Step;
END_VAR
VAR // added by the converter: edge detectors and wires of the graphical bodies
    _w1 : INT;
    _w2, _w3, _w4, _w5, _w6, _w7, _w8, _w9, _w10, _w11, _w12, _w13, _w14 : BOOL;
END_VAR

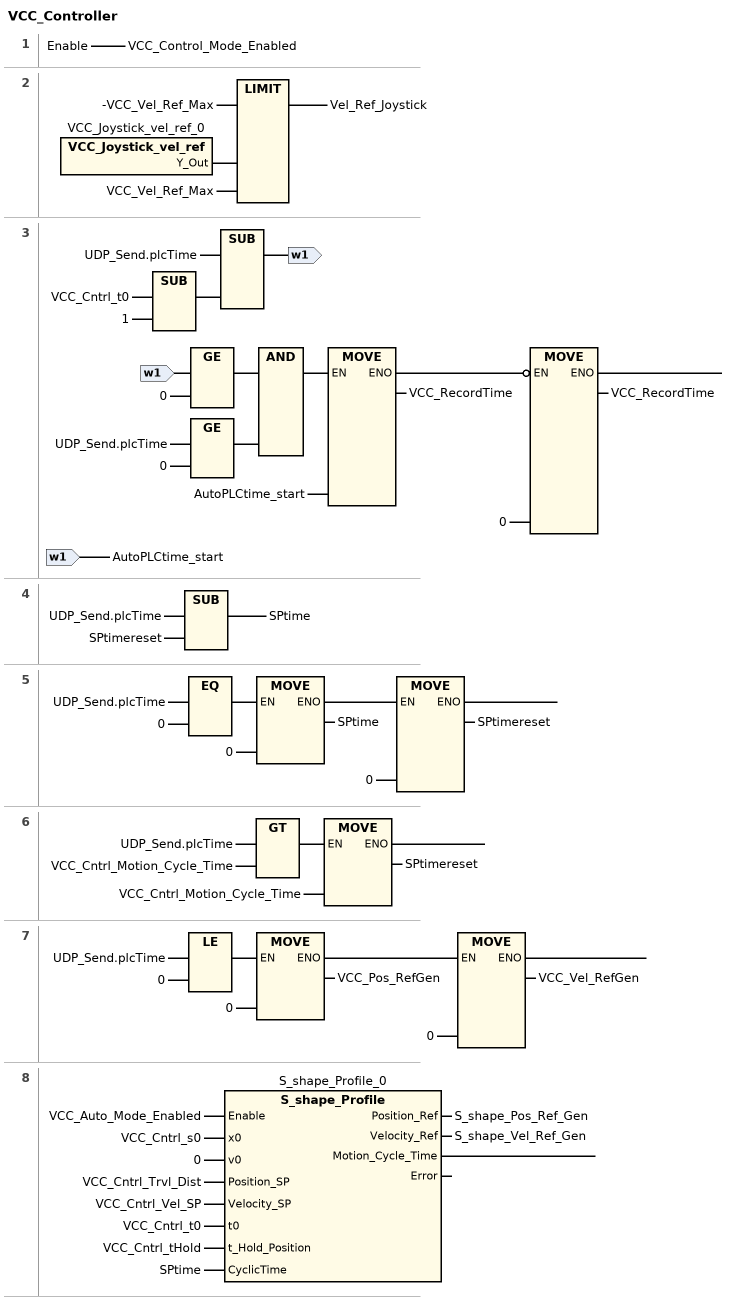
// NETWORK 1
VCC_Control_Mode_Enabled := Enable;

// NETWORK 2
VCC_Joystick_vel_ref_0(); // VCC_Joystick_vel_ref
Vel_Ref_Joystick := LIMIT(-VCC_Vel_Ref_Max, VCC_Joystick_vel_ref_0.Y_Out, VCC_Vel_Ref_Max);

// NETWORK 3
_w1 := UDP_Send.plcTime - (VCC_Cntrl_t0 - 1);
IF _w1 >= 0 AND UDP_Send.plcTime >= 0 THEN VCC_RecordTime := AutoPLCtime_start; END_IF
IF NOT (_w1 >= 0 AND UDP_Send.plcTime >= 0) THEN VCC_RecordTime := 0; END_IF
AutoPLCtime_start := _w1;

// NETWORK 4
SPtime := UDP_Send.plcTime - SPtimereset;

// NETWORK 5
_w2 := UDP_Send.plcTime = 0;
IF _w2 THEN SPtime := 0; END_IF
IF _w2 THEN SPtimereset := 0; END_IF

// NETWORK 6
IF UDP_Send.plcTime > VCC_Cntrl_Motion_Cycle_Time THEN SPtimereset := VCC_Cntrl_Motion_Cycle_Time; END_IF

// NETWORK 7
_w3 := UDP_Send.plcTime <= 0;
IF _w3 THEN VCC_Pos_RefGen := 0; END_IF
IF _w3 THEN VCC_Vel_RefGen := 0; END_IF

// NETWORK 8
S_shape_Profile_0(
    Enable := VCC_Auto_Mode_Enabled,
    x0 := VCC_Cntrl_s0,
    v0 := 0,
    Position_SP := VCC_Cntrl_Trvl_Dist,
    Velocity_SP := VCC_Cntrl_Vel_SP,
    t0 := VCC_Cntrl_t0,
    t_Hold_Position := VCC_Cntrl_tHold,
    CyclicTime := SPtime,
    Position_Ref => S_shape_Pos_Ref_Gen,
    Velocity_Ref => S_shape_Vel_Ref_Gen); // S_shape_Profile

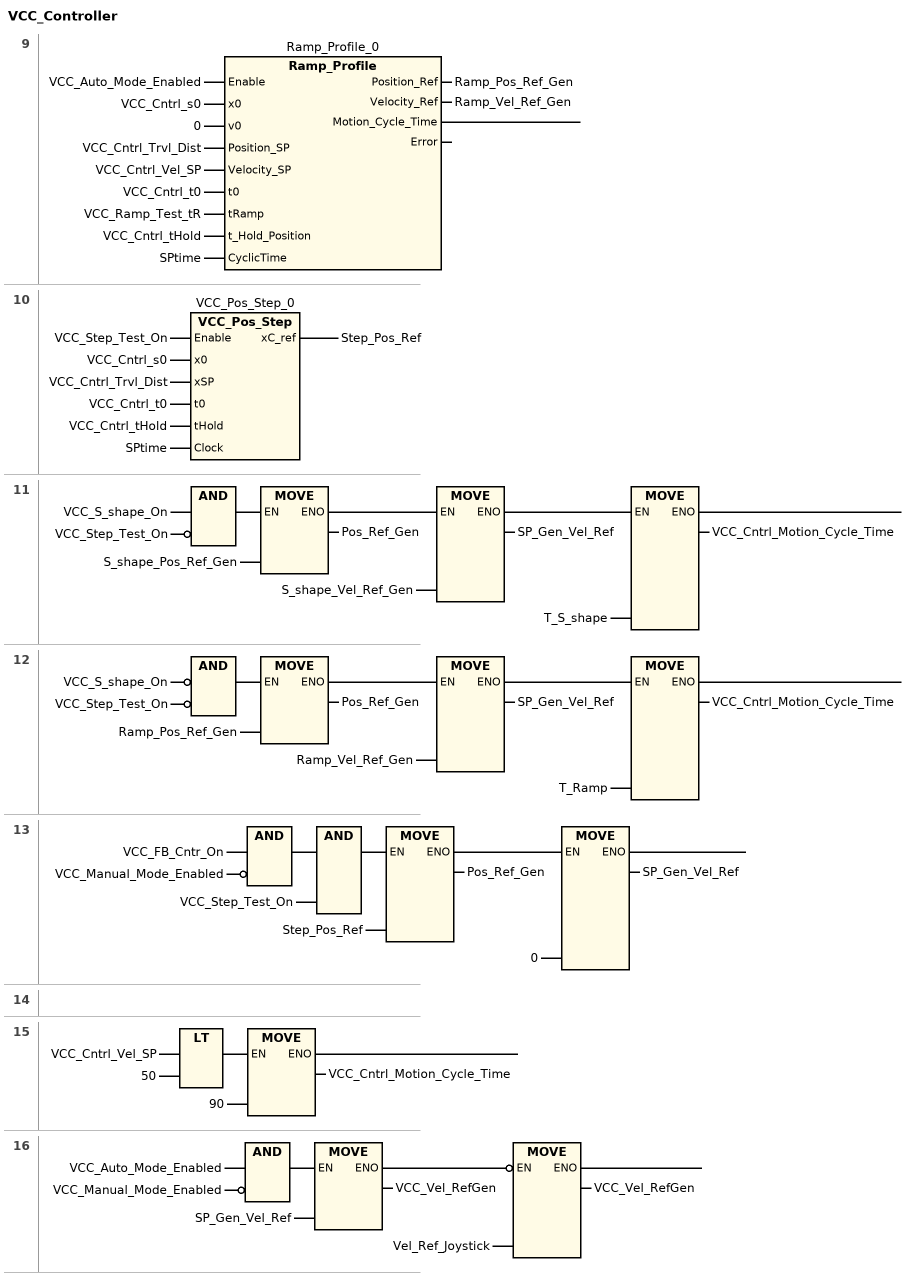
// NETWORK 9
Ramp_Profile_0(
    Enable := VCC_Auto_Mode_Enabled,
    x0 := VCC_Cntrl_s0,
    v0 := 0,
    Position_SP := VCC_Cntrl_Trvl_Dist,
    Velocity_SP := VCC_Cntrl_Vel_SP,
    t0 := VCC_Cntrl_t0,
    tRamp := VCC_Ramp_Test_tR,
    t_Hold_Position := VCC_Cntrl_tHold,
    CyclicTime := SPtime,
    Position_Ref => Ramp_Pos_Ref_Gen,
    Velocity_Ref => Ramp_Vel_Ref_Gen); // Ramp_Profile

// NETWORK 10
VCC_Pos_Step_0(
    Enable := VCC_Step_Test_On,
    x0 := VCC_Cntrl_s0,
    xSP := VCC_Cntrl_Trvl_Dist,
    t0 := VCC_Cntrl_t0,
    tHold := VCC_Cntrl_tHold,
    Clock := SPtime); // VCC_Pos_Step
Step_Pos_Ref := VCC_Pos_Step_0.xC_ref;

// NETWORK 11
_w4 := VCC_S_shape_On AND NOT VCC_Step_Test_On;
IF _w4 THEN Pos_Ref_Gen := S_shape_Pos_Ref_Gen; END_IF
IF _w4 THEN SP_Gen_Vel_Ref := S_shape_Vel_Ref_Gen; END_IF
IF _w4 THEN VCC_Cntrl_Motion_Cycle_Time := T_S_shape; END_IF

// NETWORK 12
_w5 := NOT VCC_S_shape_On AND NOT VCC_Step_Test_On;
IF _w5 THEN Pos_Ref_Gen := Ramp_Pos_Ref_Gen; END_IF
IF _w5 THEN SP_Gen_Vel_Ref := Ramp_Vel_Ref_Gen; END_IF
IF _w5 THEN VCC_Cntrl_Motion_Cycle_Time := T_Ramp; END_IF

// NETWORK 13
_w6 := (VCC_FB_Cntr_On AND NOT VCC_Manual_Mode_Enabled) AND VCC_Step_Test_On;
IF _w6 THEN Pos_Ref_Gen := Step_Pos_Ref; END_IF
IF _w6 THEN SP_Gen_Vel_Ref := 0; END_IF

// NETWORK 14

// NETWORK 15
IF VCC_Cntrl_Vel_SP < 50 THEN VCC_Cntrl_Motion_Cycle_Time := 90; END_IF

// NETWORK 16
_w7 := VCC_Auto_Mode_Enabled AND NOT VCC_Manual_Mode_Enabled;
IF _w7 THEN VCC_Vel_RefGen := SP_Gen_Vel_Ref; END_IF
IF NOT _w7 THEN VCC_Vel_RefGen := Vel_Ref_Joystick; END_IF

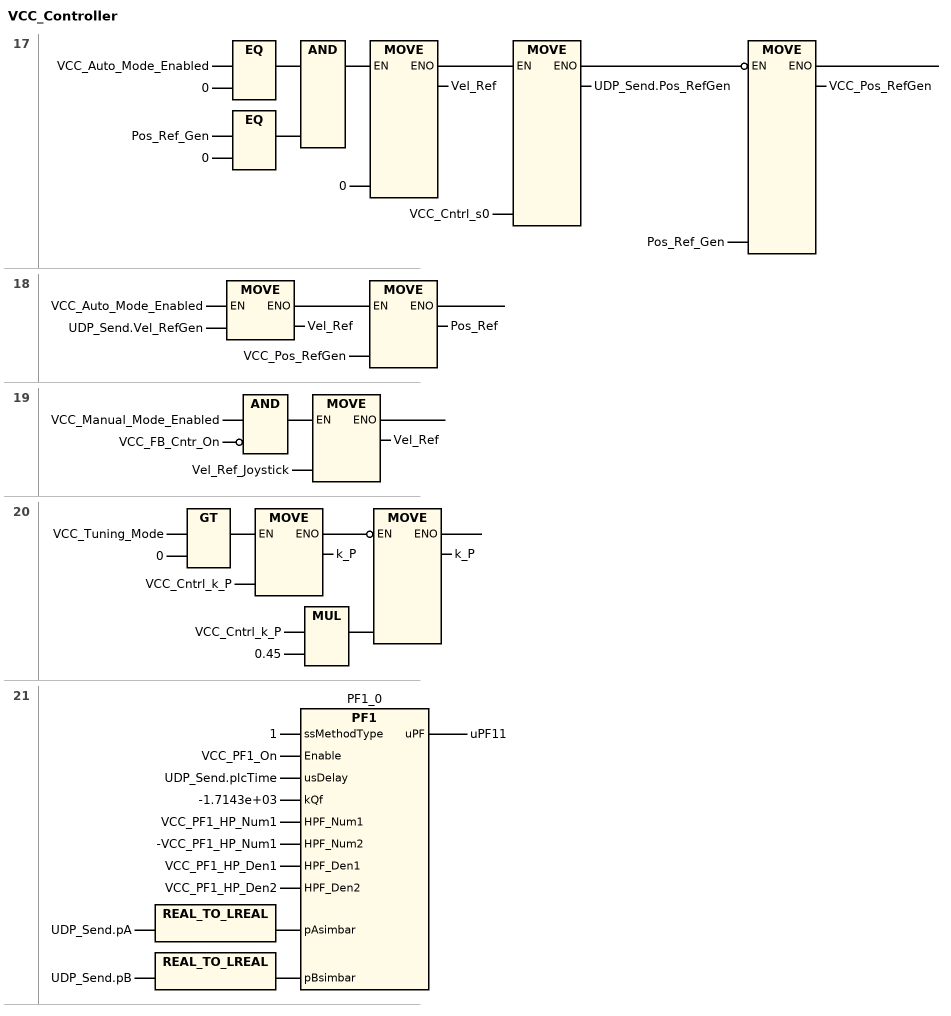
// NETWORK 17
_w8 := VCC_Auto_Mode_Enabled = 0 AND Pos_Ref_Gen = 0;
IF _w8 THEN Vel_Ref := 0; END_IF
IF _w8 THEN UDP_Send.Pos_RefGen := VCC_Cntrl_s0; END_IF
IF NOT _w8 THEN VCC_Pos_RefGen := Pos_Ref_Gen; END_IF

// NETWORK 18
_w9 := VCC_Auto_Mode_Enabled;
IF _w9 THEN Vel_Ref := UDP_Send.Vel_RefGen; END_IF
IF _w9 THEN Pos_Ref := VCC_Pos_RefGen; END_IF

// NETWORK 19
IF VCC_Manual_Mode_Enabled AND NOT VCC_FB_Cntr_On THEN Vel_Ref := Vel_Ref_Joystick; END_IF

// NETWORK 20
_w10 := VCC_Tuning_Mode > 0;
IF _w10 THEN k_P := VCC_Cntrl_k_P; END_IF
IF NOT _w10 THEN k_P := VCC_Cntrl_k_P * 0.45; END_IF

// NETWORK 21
PF1_0(
    ssMethodType := 1,
    Enable := VCC_PF1_On,
    usDelay := UDP_Send.plcTime,
    kQf := -1.7143e+03,
    HPF_Num1 := VCC_PF1_HP_Num1,
    HPF_Num2 := -VCC_PF1_HP_Num1,
    HPF_Den1 := VCC_PF1_HP_Den1,
    HPF_Den2 := VCC_PF1_HP_Den2,
    pAsimbar := REAL_TO_LREAL(UDP_Send.pA),
    pBsimbar := REAL_TO_LREAL(UDP_Send.pB)); // PF1
uPF11 := PF1_0.uPF;

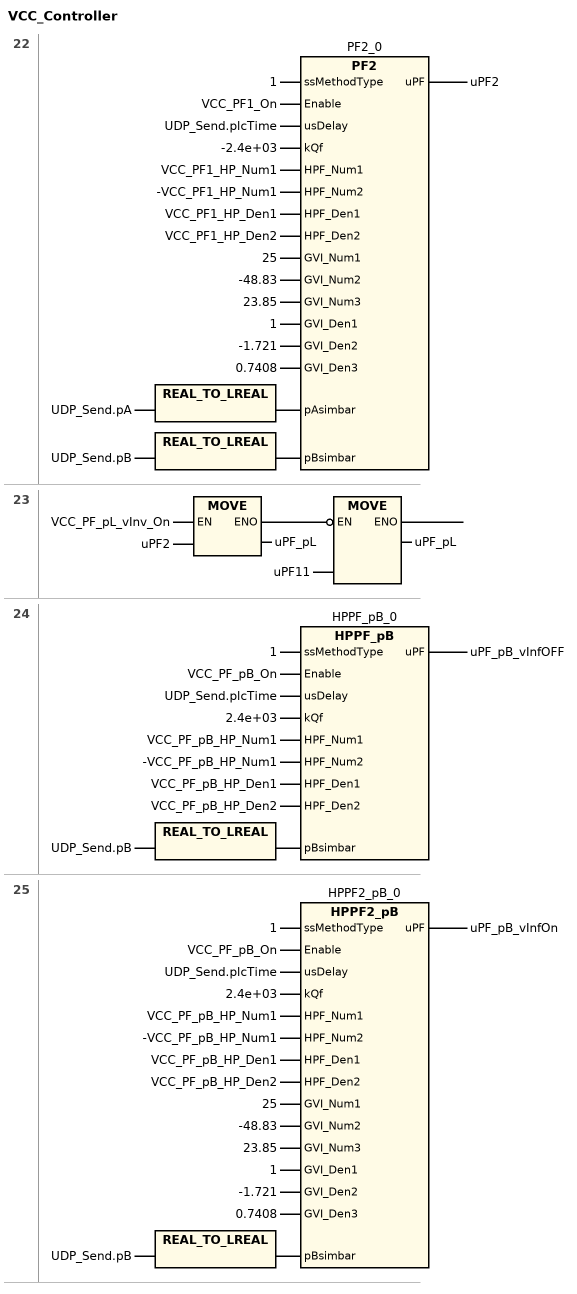
// NETWORK 22
PF2_0(
    ssMethodType := 1,
    Enable := VCC_PF1_On,
    usDelay := UDP_Send.plcTime,
    kQf := -2.4e+03,
    HPF_Num1 := VCC_PF1_HP_Num1,
    HPF_Num2 := -VCC_PF1_HP_Num1,
    HPF_Den1 := VCC_PF1_HP_Den1,
    HPF_Den2 := VCC_PF1_HP_Den2,
    GVI_Num1 := 25,
    GVI_Num2 := -48.83,
    GVI_Num3 := 23.85,
    GVI_Den1 := 1,
    GVI_Den2 := -1.721,
    GVI_Den3 := 0.7408,
    pAsimbar := REAL_TO_LREAL(UDP_Send.pA),
    pBsimbar := REAL_TO_LREAL(UDP_Send.pB)); // PF2
uPF2 := PF2_0.uPF;

// NETWORK 23
_w11 := VCC_PF_pL_vInv_On;
IF _w11 THEN uPF_pL := uPF2; END_IF
IF NOT _w11 THEN uPF_pL := uPF11; END_IF

// NETWORK 24
HPPF_pB_0(
    ssMethodType := 1,
    Enable := VCC_PF_pB_On,
    usDelay := UDP_Send.plcTime,
    kQf := 2.4e+03,
    HPF_Num1 := VCC_PF_pB_HP_Num1,
    HPF_Num2 := -VCC_PF_pB_HP_Num1,
    HPF_Den1 := VCC_PF_pB_HP_Den1,
    HPF_Den2 := VCC_PF_pB_HP_Den2,
    pBsimbar := REAL_TO_LREAL(UDP_Send.pB)); // HPPF_pB
uPF_pB_vInfOFF := HPPF_pB_0.uPF;

// NETWORK 25
HPPF2_pB_0(
    ssMethodType := 1,
    Enable := VCC_PF_pB_On,
    usDelay := UDP_Send.plcTime,
    kQf := 2.4e+03,
    HPF_Num1 := VCC_PF_pB_HP_Num1,
    HPF_Num2 := -VCC_PF_pB_HP_Num1,
    HPF_Den1 := VCC_PF_pB_HP_Den1,
    HPF_Den2 := VCC_PF_pB_HP_Den2,
    GVI_Num1 := 25,
    GVI_Num2 := -48.83,
    GVI_Num3 := 23.85,
    GVI_Den1 := 1,
    GVI_Den2 := -1.721,
    GVI_Den3 := 0.7408,
    pBsimbar := REAL_TO_LREAL(UDP_Send.pB)); // HPPF2_pB
uPF_pB_vInfOn := HPPF2_pB_0.uPF;

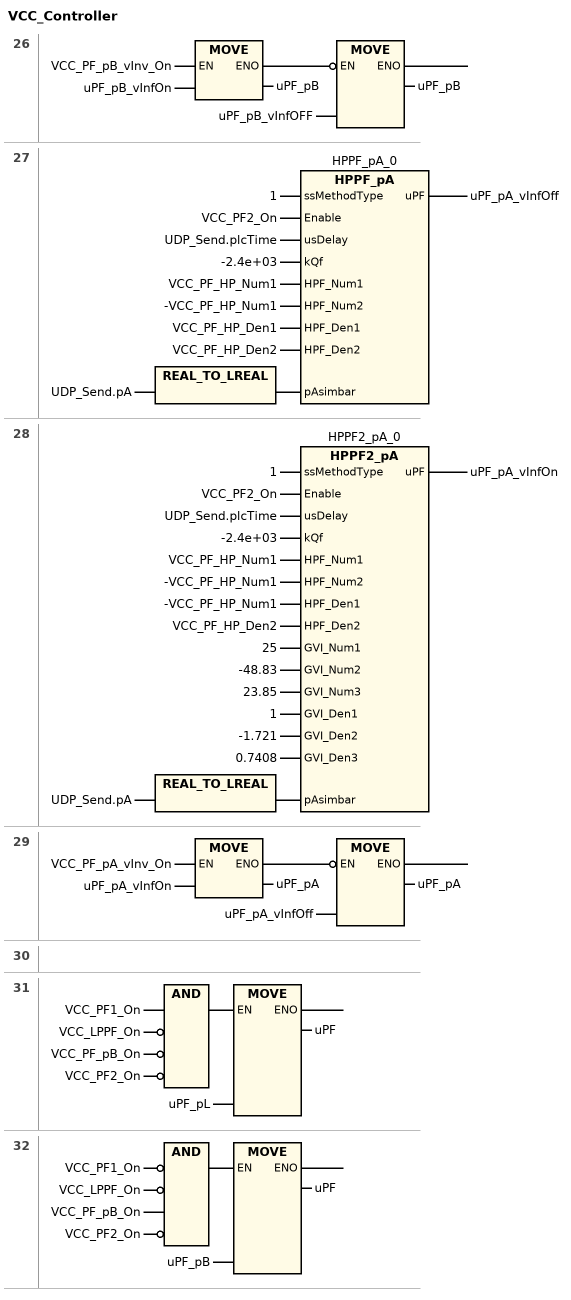
// NETWORK 26
_w12 := VCC_PF_pB_vInv_On;
IF _w12 THEN uPF_pB := uPF_pB_vInfOn; END_IF
IF NOT _w12 THEN uPF_pB := uPF_pB_vInfOFF; END_IF

// NETWORK 27
HPPF_pA_0(
    ssMethodType := 1,
    Enable := VCC_PF2_On,
    usDelay := UDP_Send.plcTime,
    kQf := -2.4e+03,
    HPF_Num1 := VCC_PF_HP_Num1,
    HPF_Num2 := -VCC_PF_HP_Num1,
    HPF_Den1 := VCC_PF_HP_Den1,
    HPF_Den2 := VCC_PF_HP_Den2,
    pAsimbar := REAL_TO_LREAL(UDP_Send.pA)); // HPPF_pA
uPF_pA_vInfOff := HPPF_pA_0.uPF;

// NETWORK 28
HPPF2_pA_0(
    ssMethodType := 1,
    Enable := VCC_PF2_On,
    usDelay := UDP_Send.plcTime,
    kQf := -2.4e+03,
    HPF_Num1 := VCC_PF_HP_Num1,
    HPF_Num2 := -VCC_PF_HP_Num1,
    HPF_Den1 := -VCC_PF_HP_Num1,
    HPF_Den2 := VCC_PF_HP_Den2,
    GVI_Num1 := 25,
    GVI_Num2 := -48.83,
    GVI_Num3 := 23.85,
    GVI_Den1 := 1,
    GVI_Den2 := -1.721,
    GVI_Den3 := 0.7408,
    pAsimbar := REAL_TO_LREAL(UDP_Send.pA)); // HPPF2_pA
uPF_pA_vInfOn := HPPF2_pA_0.uPF;

// NETWORK 29
_w13 := VCC_PF_pA_vInv_On;
IF _w13 THEN uPF_pA := uPF_pA_vInfOn; END_IF
IF NOT _w13 THEN uPF_pA := uPF_pA_vInfOff; END_IF

// NETWORK 30

// NETWORK 31
IF VCC_PF1_On AND NOT VCC_LPPF_On AND NOT VCC_PF_pB_On AND NOT VCC_PF2_On THEN uPF := uPF_pL; END_IF

// NETWORK 32
IF NOT VCC_PF1_On AND NOT VCC_LPPF_On AND VCC_PF_pB_On AND NOT VCC_PF2_On THEN uPF := uPF_pB; END_IF

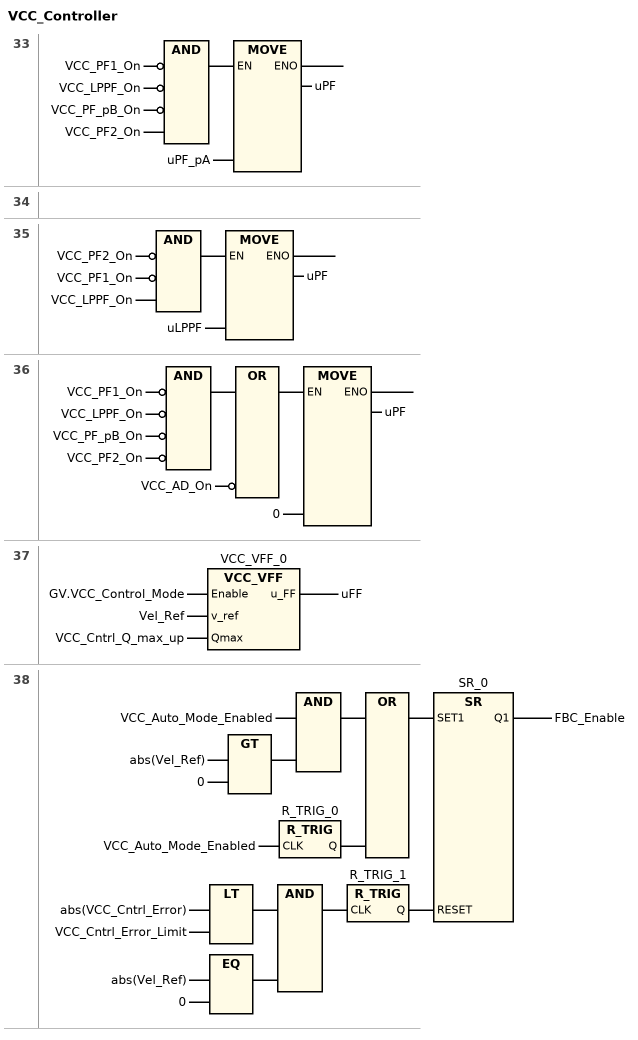
// NETWORK 33
IF NOT VCC_PF1_On AND NOT VCC_LPPF_On AND NOT VCC_PF_pB_On AND VCC_PF2_On THEN uPF := uPF_pA; END_IF

// NETWORK 34

// NETWORK 35
IF NOT VCC_PF2_On AND NOT VCC_PF1_On AND VCC_LPPF_On THEN uPF := uLPPF; END_IF

// NETWORK 36
IF NOT VCC_PF1_On AND NOT VCC_LPPF_On AND NOT VCC_PF_pB_On AND NOT VCC_PF2_On OR NOT VCC_AD_On THEN
    uPF := 0;
END_IF

// NETWORK 37
VCC_VFF_0(Enable := GV.VCC_Control_Mode, v_ref := Vel_Ref, Qmax := VCC_Cntrl_Q_max_up); // VCC_VFF
uFF := VCC_VFF_0.u_FF;

// NETWORK 38
R_TRIG_0(CLK := VCC_Auto_Mode_Enabled); // R_TRIG
R_TRIG_1(CLK := (abs(VCC_Cntrl_Error)) < VCC_Cntrl_Error_Limit AND (abs(Vel_Ref)) = 0); // R_TRIG
SR_0(SET1 := VCC_Auto_Mode_Enabled AND (abs(Vel_Ref)) > 0 OR R_TRIG_0.Q, RESET := R_TRIG_1.Q); // SR
FBC_Enable := SR_0.Q1;

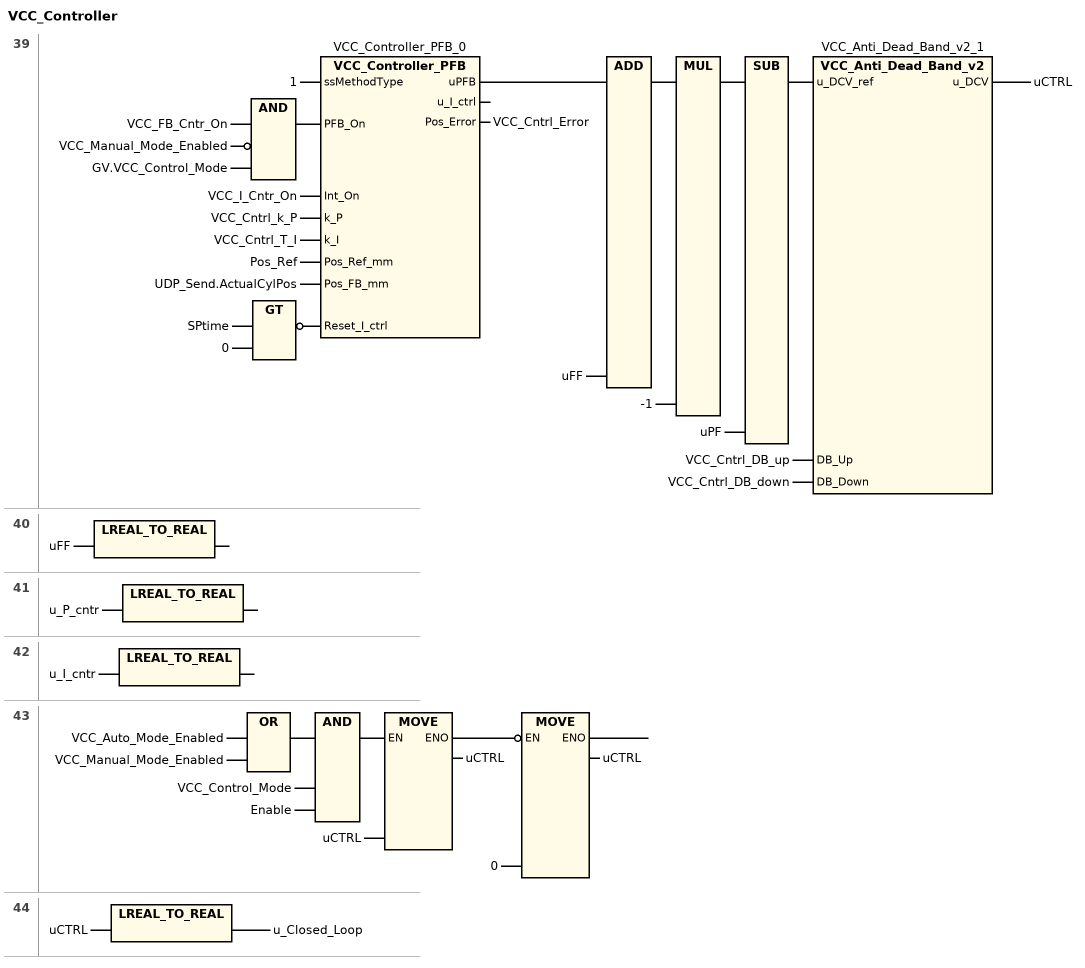
// NETWORK 39
VCC_Controller_PFB_0(
    ssMethodType := 1,
    PFB_On := VCC_FB_Cntr_On AND NOT VCC_Manual_Mode_Enabled AND GV.VCC_Control_Mode,
    Int_On := VCC_I_Cntr_On,
    k_P := VCC_Cntrl_k_P,
    k_I := VCC_Cntrl_T_I,
    Pos_Ref_mm := Pos_Ref,
    Pos_FB_mm := UDP_Send.ActualCylPos,
    Reset_I_ctrl := NOT (SPtime > 0),
    Pos_Error => VCC_Cntrl_Error); // VCC_Controller_PFB
VCC_Anti_Dead_Band_v2_1(
    u_DCV_ref := (VCC_Controller_PFB_0.uPFB + uFF) * -1 - uPF,
    DB_Up := VCC_Cntrl_DB_up,
    DB_Down := VCC_Cntrl_DB_down); // VCC_Anti_Dead_Band_v2
uCTRL := VCC_Anti_Dead_Band_v2_1.u_DCV;

// NETWORK 40
LREAL_TO_REAL(uFF);

// NETWORK 41
LREAL_TO_REAL(u_P_cntr);

// NETWORK 42
LREAL_TO_REAL(u_I_cntr);

// NETWORK 43
_w14 := (VCC_Auto_Mode_Enabled OR VCC_Manual_Mode_Enabled) AND VCC_Control_Mode AND Enable;
IF _w14 THEN uCTRL := uCTRL; END_IF
IF NOT _w14 THEN uCTRL := 0; END_IF

// NETWORK 44
u_Closed_Loop := LREAL_TO_REAL(uCTRL);

END_PROGRAM

// IndraMotionMlc1/Application/VCC_VFF
FUNCTION_BLOCK VCC_VFF
VAR_INPUT
	Enable: BOOL;
	v_ref: LREAL;
	Qmax: LREAL;
END_VAR
VAR_OUTPUT
	u_FF: LREAL;
END_VAR
VAR
	rtb_Switch1: LREAL;
END_VAR


(* Switch: '<S1>/Switch2' incorporates:
 *  Constant: '<S1>/Annnulus_Area'
 *  Constant: '<S1>/Bore_Area'
 *  Product: '<S1>/Product1'
 *  Product: '<S1>/Product3' *)

IF v_ref >= 0.0 THEN 
    rtb_Switch1 := 3318.3 * v_ref;
ELSE 
    rtb_Switch1 := v_ref * 2356.2;
END_IF;

(* End of Switch: '<S1>/Switch2' *)


(* Switch: '<S1>/Switch1' *)

IF Enable THEN 
    (* Outport: '<Root>/u_FF [-]' incorporates:
     *  Gain: '<S1>/Gain1'
     *  Gain: '<S1>/Gain3'
     *  Product: '<S1>/Divide2' *)
    u_FF := ((1.0E-9 * rtb_Switch1) * 60000.0) / Qmax;
ELSE 
    (* Outport: '<Root>/u_FF [-]' incorporates:
     *  Constant: '<S1>/Constant' *)
    u_FF := 0.0;
END_IF;

(* End of Switch: '<S1>/Switch1' *)

END_FUNCTION_BLOCK

// IndraMotionMlc1/Application/VCC_Controller_PFB
FUNCTION_BLOCK VCC_Controller_PFB
VAR_INPUT
	ssMethodType: SINT;
	PFB_On: BOOL;
	Int_On: BOOL;
	k_P: LREAL;
	k_I: LREAL;
	Pos_Ref_mm: LREAL;
	Pos_FB_mm: LREAL;
	Reset_I_ctrl: BOOL;
END_VAR
VAR_OUTPUT
	uPFB: LREAL;
	u_I_ctrl: LREAL;
	Pos_Error: LREAL;
END_VAR
VAR
	rtb_Switch2: LREAL;
	rtb_u_FB: LREAL;
	c_DiscreteTimeIntegrator_DS: LREAL;
END_VAR



CASE ssMethodType OF
    0: 
        (* InitializeConditions for DiscreteIntegrator: '<S1>/Discrete-Time Integrator' *)
        c_DiscreteTimeIntegrator_DS := 0.0;
    1: 
        (* Switch: '<S1>/Switch2' *)

        IF Reset_I_ctrl THEN 
            (* DiscreteIntegrator: '<S1>/Discrete-Time Integrator' *)
            c_DiscreteTimeIntegrator_DS := 0.0;
        END_IF;

        (* End of Switch: '<S1>/Switch2' *)
        

        (* Sum: '<S1>/Sum1' incorporates:
         *  Gain: '<S1>/Gain1'
         *  Gain: '<S1>/Gain2' *)
        rtb_Switch2 := (0.001 * Pos_Ref_mm) - (0.001 * Pos_FB_mm);
        (* Switch: '<S1>/Switch' incorporates:
         *  Constant: '<S1>/Constant'
         *  DiscreteIntegrator: '<S1>/Discrete-Time Integrator' *)

        IF Int_On THEN 
            u_I_ctrl := c_DiscreteTimeIntegrator_DS;
        ELSE 
            u_I_ctrl := 0.0;
        END_IF;

        (* End of Switch: '<S1>/Switch' *)
        

        (* Sum: '<S1>/Sum5' incorporates:
         *  Product: '<S1>/Product' *)
        rtb_u_FB := (k_P * rtb_Switch2) + u_I_ctrl;
        (* Saturate: '<S1>/Saturation1' *)

        IF rtb_u_FB >= 1.0 THEN 
            uPFB := 1.0;
        ELSIF rtb_u_FB > -1.0 THEN 
            uPFB := rtb_u_FB;
        ELSE 
            uPFB := -1.0;
        END_IF;

        (* End of Saturate: '<S1>/Saturation1' *)
        

        (* Sum: '<S1>/Sum3' *)
        rtb_u_FB := uPFB - rtb_u_FB;
        (* Switch: '<S1>/Switch1' incorporates:
         *  Constant: '<S1>/Constant1' *)

        IF  NOT PFB_On THEN 
            uPFB := 0.0;
        END_IF;

        (* End of Switch: '<S1>/Switch1' *)
        

        (* Outport: '<Root>/Pos_Error' incorporates:
         *  Gain: '<S1>/Gain3' *)
        Pos_Error := -1000.0 * rtb_Switch2;
        (* Update for DiscreteIntegrator: '<S1>/Discrete-Time Integrator' incorporates:
         *  Product: '<S1>/Divide'
         *  Product: '<S1>/Product2'
         *  Sum: '<S1>/Sum2' *)
        c_DiscreteTimeIntegrator_DS := ((((rtb_u_FB / k_P) + rtb_Switch2) * k_I) * 0.001) + c_DiscreteTimeIntegrator_DS;
END_CASE;

END_FUNCTION_BLOCK

// IndraMotionMlc1/Application/VCC_PI_Controller
FUNCTION_BLOCK VCC_PI_Controller
VAR_INPUT
	ssMethodType: SINT;
	FB_Cntr_On: LREAL;
	I_Cntr_On: LREAL;
	k_P: LREAL;
	k_I: LREAL;
	I_Cntr_Reset: LREAL;
	FeedForward: LREAL;
	Pos_Ref: LREAL;
	Pos_FB: LREAL;
END_VAR
VAR_OUTPUT
	Pos_Error: LREAL;
	uFB: LREAL;
	uFF: LREAL;
	uSignal: LREAL;
END_VAR
VAR
	rtb_Sum3: LREAL;
	c_DiscreteTimeIntegrator_DS: LREAL;
END_VAR



CASE ssMethodType OF
    0: 
        (* InitializeConditions for DiscreteIntegrator: '<S1>/Discrete-Time Integrator' *)
        c_DiscreteTimeIntegrator_DS := 0.0;
    1: 
        (* DiscreteIntegrator: '<S1>/Discrete-Time Integrator' *)

        IF I_Cntr_Reset <> 0.0 THEN 
            c_DiscreteTimeIntegrator_DS := 0.0;
        END_IF;

        (* Sum: '<S1>/Sum1' *)
        Pos_Error := Pos_Ref - Pos_FB;
        (* Switch: '<S1>/Switch' incorporates:
         *  Constant: '<S1>/Constant'
         *  DiscreteIntegrator: '<S1>/Discrete-Time Integrator' *)

        IF I_Cntr_On > 0.0 THEN 
            uSignal := c_DiscreteTimeIntegrator_DS;
        ELSE 
            uSignal := 0.0;
        END_IF;

        (* End of Switch: '<S1>/Switch' *)
        

        (* Sum: '<S1>/Sum' incorporates:
         *  Product: '<S1>/Product' *)
        uSignal := (k_P * Pos_Error) + uSignal;
        (* Saturate: '<S1>/Saturation' *)

        IF uSignal >= 1.0 THEN 
            uFB := 1.0;
        ELSIF uSignal > -1.0 THEN 
            uFB := uSignal;
        ELSE 
            uFB := -1.0;
        END_IF;

        (* End of Saturate: '<S1>/Saturation' *)
        

        (* Sum: '<S1>/Sum3' *)
        rtb_Sum3 := uFB - uSignal;
        (* Switch: '<S1>/Switch1' incorporates:
         *  Constant: '<S1>/Constant1' *)

        IF  NOT (FB_Cntr_On > 0.0) THEN 
            uFB := 0.0;
        END_IF;

        (* End of Switch: '<S1>/Switch1' *)
        

        (* Sum: '<S1>/Sum4' *)
        uSignal := FeedForward + uFB;
        (* Saturate: '<S1>/Saturation1' *)

        IF uSignal >= 1.0 THEN 
            (* Outport: '<Root>/uSignal' *)
            uSignal := 1.0;
        ELSIF  NOT (uSignal > -1.0) THEN 
            (* Outport: '<Root>/uSignal' *)
            uSignal := -1.0;
        END_IF;

        (* End of Saturate: '<S1>/Saturation1' *)
        

        (* Outport: '<Root>/uFF' *)
        uFF := FeedForward;
        (* Update for DiscreteIntegrator: '<S1>/Discrete-Time Integrator' incorporates:
         *  Product: '<S1>/Divide'
         *  Product: '<S1>/Product2'
         *  Sum: '<S1>/Sum2' *)
        c_DiscreteTimeIntegrator_DS := ((((rtb_Sum3 / k_P) + Pos_Error) * k_I) * 0.001) + c_DiscreteTimeIntegrator_DS;
END_CASE;

END_FUNCTION_BLOCK

// IndraMotionMlc1/Application/VCC_Controller_FF_PI_AD_v05
FUNCTION_BLOCK VCC_Controller_FF_PI_AD_v05
VAR_INPUT
	ssMethodType: SINT;
	Tuning_Mode_On: BOOL;
	FF_Valve_Mapping_On: BOOL;
	FB_Cntr_On: BOOL;
	I_Cntr_On: BOOL;
	I_Cntr_Reset_On: BOOL;
	Active_Damper_On: BOOL;
	k_AD_Num: LREAL;
	Pos_Error_Limit: LREAL;
	DB_Up: LREAL;
	DB_Down: LREAL;
	Qmax_Up: LREAL;
	Qmax_Down: LREAL;
	k_P: LREAL;
	k_I: LREAL;
	Pos_Ref: LREAL;
	Vel_Ref: LREAL;
	Pos_FB: LREAL;
	p_A: LREAL;
	p_B: LREAL;
END_VAR
VAR_OUTPUT
	Pos_Error: LREAL;
	u_FF: LREAL;
	u_P: LREAL;
	u_I: LREAL;
	u_AD: LREAL;
	I_reset: LREAL;
	u_DCV: LREAL;
END_VAR
VAR
	iRght: UDINT;
	iLeft: UDINT;
	bpIdx: UDINT;
	rtb_u_ref: LREAL;
	rtb_Saturation1: LREAL;
	rtb_I_Reset: LREAL;
	rtb_LoadPressure: LREAL;
	c_DiscreteTimeIntegrator_DS: LREAL;
	VectorConcatenate: ARRAY[0..1] OF LREAL;
	TransferFcn11_states: LREAL;
	uvsQValve2_bp01Data: ARRAY[0..34] OF LREAL := [-64.5, -64.49, -61.0, -56.5, -52.5, -47.0, -41.9, -36.0, -29.6, -23.5, -17.3, -11.7, -7.2, -3.3, -0.9, -0.5, -0.1, -1.0E-10, 0.0, 1.0E-10, 0.1, 0.8, 5.0, 10.8, 16.5, 23.0, 31.0, 38.5, 44.8, 49.7, 55.0, 60.0, 65.498, 65.499, 65.5];
	uvsQValve2_tableData: ARRAY[0..34] OF LREAL := [1.0, 0.95, 0.9, 0.85, 0.8, 0.75, 0.7, 0.65, 0.6, 0.55, 0.5, 0.45, 0.4, 0.35, 0.3, 0.25, 0.236, 0.2359999999, 0.0, -0.32999999999999, -0.33, -0.35, -0.4, -0.45, -0.5, -0.55, -0.6, -0.65, -0.7, -0.75, -0.8, -0.85, -0.9, -0.95, -1.0];
END_VAR



CASE ssMethodType OF
    0: 
        (* InitializeConditions for DiscreteIntegrator: '<S1>/Discrete-Time Integrator' *)
        c_DiscreteTimeIntegrator_DS := 0.0;
        (* InitializeConditions for DiscreteTransferFcn: '<S5>/Transfer Fcn1 1' *)
        TransferFcn11_states := 0.0;
    1: 
        (* Switch: '<S1>/Switch2' incorporates:
         *  Constant: '<S1>/Annnulus_Area'
         *  Constant: '<S1>/Bore_Area'
         *  Product: '<S1>/Product1'
         *  Product: '<S1>/Product3' *)

        IF Vel_Ref >= 0.0 THEN 
            u_AD := 3318.3 * Vel_Ref;
        ELSE 
            u_AD := Vel_Ref * 2356.2;
        END_IF;

        (* End of Switch: '<S1>/Switch2' *)
        

        (* Gain: '<S1>/Gain1' incorporates:
         *  Gain: '<S1>/Gain2' *)
        u_AD := (1.0E-9 * u_AD) * 60000.0;
        (* Lookup_n-D: '<S1>/ u vs Q [Valve#2]' *)
        (* Lookup 1-D
           Search method: 'binary'
           Use previous index: 'off'
           Interpolation method: 'Linear'
           Extrapolation method: 'Linear'
           Use last breakpoint for index at or above upper limit: 'off'
           Remove protection against out-of-range input in generated code: 'off' *)
        (* Prelookup - Index and Fraction
           Index Search method: 'binary'
           Extrapolation method: 'Linear'
           Use previous index: 'off'
           Use last breakpoint for index at or above upper limit: 'off'
           Remove protection against out-of-range input in generated code: 'off' *)

        IF u_AD <= -64.5 THEN 
            iLeft := 0;
            rtb_I_Reset := (u_AD - -64.5) / 0.010000000000005116;
        ELSIF u_AD < 65.5 THEN 
            (* Binary Search *)
            bpIdx := 17;
            iLeft := 0;
            iRght := 34;
            WHILE (iRght - iLeft) > 1 DO

                IF u_AD < uvsQValve2_bp01Data[bpIdx] THEN 
                    iRght := bpIdx;
                ELSE 
                    iLeft := bpIdx;
                END_IF;

                bpIdx := DWORD_TO_UDINT(SHR(UDINT_TO_DWORD(iRght + iLeft), 1));
            END_WHILE;
            rtb_I_Reset := (u_AD - uvsQValve2_bp01Data[iLeft]) / (uvsQValve2_bp01Data[iLeft + 1] - uvsQValve2_bp01Data[iLeft]);
        ELSE 
            iLeft := 33;
            rtb_I_Reset := (u_AD - 65.499) / 0.0010000000000047748;
        END_IF;

        (* Switch: '<S1>/Switch5' *)
        (* Interpolation 1-D
           Interpolation method: 'Linear'
           Use last breakpoint for index at or above upper limit: 'off'
           Overflow mode: 'wrapping' *)

        IF Vel_Ref >= 0.0 THEN 
            u_FF := Qmax_Up;
        ELSE 
            u_FF := Qmax_Down;
        END_IF;

        (* End of Switch: '<S1>/Switch5' *)
        

        (* Product: '<S1>/Divide2' *)
        rtb_u_ref := u_AD / u_FF;
        (* MATLAB Function: '<S1>/AntiDB' *)
        (* MATLAB Function 'VCC_Controller_FF_PI_AD_v05/AntiDB': '<S2>:1' *)
        (* '<S2>:1:5' u_DCV = 0; *)
        (* '<S2>:1:8' if (u_DCV_ref < -0.001) *)

        IF rtb_u_ref < -0.001 THEN 
            (* '<S2>:1:9' u_DCV = -DB_Up + (1-DB_Up)*u_DCV_ref; *)
            u_FF := ((1.0 - DB_Up) * rtb_u_ref) + ( -DB_Up);
        ELSIF rtb_u_ref > 0.001 THEN 
            (* '<S2>:1:10' elseif (u_DCV_ref > 0.001) *)
            (* '<S2>:1:11' u_DCV = DB_Down + (1-DB_Down)*u_DCV_ref; *)
            u_FF := ((1.0 - DB_Down) * rtb_u_ref) + DB_Down;
        ELSE 
            (* '<S2>:1:12' else *)
            (* '<S2>:1:13' u_DCV = 0; *)
            u_FF := 0.0;
        END_IF;

        (* End of MATLAB Function: '<S1>/AntiDB' *)
        

        (* Switch: '<S1>/Switch6' incorporates:
         *  Gain: '<S1>/Gain3'
         *  Lookup_n-D: '<S1>/ u vs Q [Valve#2]' *)

        IF FF_Valve_Mapping_On THEN 
            u_FF :=  -(((uvsQValve2_tableData[iLeft + 1] - uvsQValve2_tableData[iLeft]) * rtb_I_Reset) + uvsQValve2_tableData[iLeft]);
        END_IF;

        (* End of Switch: '<S1>/Switch6' *)
        

        (* Sum: '<S1>/Sum1' *)
        Pos_Error := Pos_Ref - Pos_FB;
        (* Product: '<S1>/Product' *)
        u_P := k_P * Pos_Error;
        (* MATLAB Function: '<S1>/Controller_Reset' *)
        (* MATLAB Function 'VCC_Controller_FF_PI_AD_v05/Controller_Reset': '<S4>:1' *)
        (* '<S4>:1:3' I_Reset = 1; *)
        (* '<S4>:1:5' if (abs(Pos_Error) <= Pos_Error_Limit) &amp;&amp; (Vel_SP == 0) *)

        IF ABS(Pos_Error) <= Pos_Error_Limit THEN 

            IF Vel_Ref = 0.0 THEN 
                (* '<S4>:1:6' I_Reset = 1; *)
                rtb_I_Reset := 1.0;
            ELSE 
                (* '<S4>:1:7' else *)
                (* '<S4>:1:8' I_Reset = 0; *)
                rtb_I_Reset := 0.0;
            END_IF;

        ELSE 
            (* '<S4>:1:7' else *)
            (* '<S4>:1:8' I_Reset = 0; *)
            rtb_I_Reset := 0.0;
        END_IF;

        (* End of MATLAB Function: '<S1>/Controller_Reset' *)
        

        (* Switch: '<S1>/Switch3' incorporates:
         *  Constant: '<S1>/Constant2' *)

        IF I_Cntr_Reset_On THEN 
            I_reset := rtb_I_Reset;
        ELSE 
            I_reset := 0.0;
        END_IF;

        (* End of Switch: '<S1>/Switch3' *)
        

        (* DiscreteIntegrator: '<S1>/Discrete-Time Integrator' *)

        IF I_reset <> 0.0 THEN 
            c_DiscreteTimeIntegrator_DS := 0.0;
        END_IF;

        (* SignalConversion: '<S5>/ConcatBufferAtVector ConcatenateIn1' *)
        VectorConcatenate[0] := k_AD_Num;
        (* Gain: '<S5>/Gain1' *)
        VectorConcatenate[1] :=  -k_AD_Num;
        (* DiscreteTransferFcn: '<S5>/Transfer Fcn1 1' incorporates:
         *  Gain: '<S5>/Cylinder Area Ratio'
         *  Sum: '<S5>/Load Pressure' *)
        rtb_u_ref := (p_A - (0.710059171597633 * p_B)) - (-0.997 * TransferFcn11_states);
        u_AD := (VectorConcatenate[0] * rtb_u_ref) + (VectorConcatenate[1] * TransferFcn11_states);
        (* Switch: '<S1>/Switch' incorporates:
         *  Constant: '<S1>/Constant'
         *  DiscreteIntegrator: '<S1>/Discrete-Time Integrator' *)

        IF I_Cntr_On THEN 
            u_I := c_DiscreteTimeIntegrator_DS;
        ELSE 
            u_I := 0.0;
        END_IF;

        (* End of Switch: '<S1>/Switch' *)
        

        (* Switch: '<S1>/Switch1' incorporates:
         *  Constant: '<S1>/Constant1'
         *  Sum: '<S1>/Sum5' *)

        IF FB_Cntr_On THEN 
            rtb_LoadPressure := u_P + u_I;
        ELSE 
            rtb_LoadPressure := 0.0;
        END_IF;

        (* End of Switch: '<S1>/Switch1' *)
        

        (* Saturate: '<S1>/Saturation1' *)

        IF rtb_LoadPressure >= 1.0 THEN 
            rtb_Saturation1 := 1.0;
        ELSIF rtb_LoadPressure > -1.0 THEN 
            rtb_Saturation1 := rtb_LoadPressure;
        ELSE 
            rtb_Saturation1 := -1.0;
        END_IF;

        (* End of Saturate: '<S1>/Saturation1' *)
        

        (* Switch: '<S1>/Switch4' incorporates:
         *  Constant: '<S1>/Constant3' *)

        IF  NOT Active_Damper_On THEN 
            u_AD := 0.0;
        END_IF;

        (* End of Switch: '<S1>/Switch4' *)
        

        (* Gain: '<S1>/Gain' incorporates:
         *  Sum: '<S1>/Sum6' *)
        u_DCV :=  -((u_FF + rtb_Saturation1) - u_AD);
        (* Saturate: '<S1>/Saturation5' *)

        IF u_DCV >= 1.0 THEN 
            u_DCV := 1.0;
        ELSIF  NOT (u_DCV > -1.0) THEN 
            u_DCV := -1.0;
        END_IF;

        (* End of Saturate: '<S1>/Saturation5' *)
        

        (* MATLAB Function: '<S1>/Anti_Dead_Band' *)
        (* MATLAB Function 'VCC_Controller_FF_PI_AD_v05/Anti_Dead_Band': '<S3>:1' *)
        (* '<S3>:1:5' u_DCV = 0; *)
        (* '<S3>:1:7' if  (I_Reset == 1) &amp;&amp; (Tuning_Mode == 0) *)

        IF (rtb_I_Reset = 1.0) AND ( NOT Tuning_Mode_On) THEN 
            (* Outport: '<Root>/u_DCV' *)
            (* '<S3>:1:8' u_DCV = 0; *)
            u_DCV := 0.0;
        END_IF;

        (* End of MATLAB Function: '<S1>/Anti_Dead_Band' *)
        

        (* Update for DiscreteIntegrator: '<S1>/Discrete-Time Integrator' incorporates:
         *  Product: '<S1>/Divide'
         *  Product: '<S1>/Product2'
         *  Sum: '<S1>/Sum2'
         *  Sum: '<S1>/Sum3' *)
        c_DiscreteTimeIntegrator_DS := (((((rtb_Saturation1 - rtb_LoadPressure) / k_P) + Pos_Error) * k_I) * 0.001) + c_DiscreteTimeIntegrator_DS;
        (* Update for DiscreteTransferFcn: '<S5>/Transfer Fcn1 1' *)
        TransferFcn11_states := rtb_u_ref;
END_CASE;

END_FUNCTION_BLOCK

// IndraMotionMlc1/Application/VCC_Controller_FF_PI_AD
FUNCTION_BLOCK VCC_Controller_FF_PI_AD
VAR_INPUT
	ssMethodType: SINT;
	Tuning_Mode_On: BOOL;
	FB_Cntr_On: BOOL;
	I_Cntr_On: BOOL;
	I_Cntr_Reset_On: BOOL;
	Active_Damper_On: BOOL;
	k_AD_Num: LREAL;
	Pos_Error_Limit: LREAL;
	DB_Up: LREAL;
	DB_Down: LREAL;
	Q_max: LREAL;
	k_P: LREAL;
	k_I: LREAL;
	Pos_Ref: LREAL;
	Vel_Ref: LREAL;
	Pos_FB: LREAL;
	p_A: LREAL;
	p_B: LREAL;
END_VAR
VAR_OUTPUT
	Pos_Error: LREAL;
	u_FF: LREAL;
	u_P: LREAL;
	u_I: LREAL;
	u_AD: LREAL;
	I_reset: LREAL;
	u_DCV: LREAL;
END_VAR
VAR
	rtb_Saturation1: LREAL;
	rtb_Gain: LREAL;
	rtb_I_Reset: DINT;
	rtb_LoadPressure: LREAL;
	TransferFcn11_tmp: LREAL;
	c_DiscreteTimeIntegrator_DS: LREAL;
	VectorConcatenate: ARRAY[0..1] OF LREAL;
	TransferFcn11_states: LREAL;
END_VAR



CASE ssMethodType OF
    0: 
        (* InitializeConditions for DiscreteIntegrator: '<S1>/Discrete-Time Integrator' *)
        c_DiscreteTimeIntegrator_DS := 0.0;
        (* InitializeConditions for DiscreteTransferFcn: '<S4>/Transfer Fcn1 1' *)
        TransferFcn11_states := 0.0;
    1: 
        (* Switch: '<S1>/Switch2' incorporates:
         *  Constant: '<S1>/Annnulus_Area'
         *  Constant: '<S1>/Bore_Area'
         *  Product: '<S1>/Product1'
         *  Product: '<S1>/Product3' *)

        IF Vel_Ref >= 0.0 THEN 
            u_FF := 3318.3 * Vel_Ref;
        ELSE 
            u_FF := Vel_Ref * 2356.2;
        END_IF;

        (* End of Switch: '<S1>/Switch2' *)
        

        (* Product: '<S1>/Divide2' incorporates:
         *  Constant: '<S1>/Constant7'
         *  Gain: '<S1>/Gain1'
         *  Gain: '<S1>/Gain2' *)
        u_FF := ((1.0E-9 * u_FF) * 60000.0) / Q_max;
        (* Sum: '<S1>/Sum1' *)
        Pos_Error := Pos_Ref - Pos_FB;
        (* Product: '<S1>/Product' *)
        u_P := k_P * Pos_Error;
        (* MATLAB Function: '<S1>/From Jespers SimX1' *)
        (* MATLAB Function 'VCC_Controller_FF_PI_AD1/From Jespers SimX1': '<S3>:1' *)
        (* '<S3>:1:3' I_Reset = 1; *)
        (* '<S3>:1:5' if (abs(Pos_Error) <= Pos_Error_Limit) &amp;&amp; (Vel_SP == 0) *)

        IF ABS(Pos_Error) <= Pos_Error_Limit THEN 

            IF Vel_Ref = 0.0 THEN 
                (* '<S3>:1:6' I_Reset = 1; *)
                rtb_I_Reset := 1;
            ELSE 
                (* '<S3>:1:7' else *)
                (* '<S3>:1:8' I_Reset = 0; *)
                rtb_I_Reset := 0;
            END_IF;

        ELSE 
            (* '<S3>:1:7' else *)
            (* '<S3>:1:8' I_Reset = 0; *)
            rtb_I_Reset := 0;
        END_IF;

        (* End of MATLAB Function: '<S1>/From Jespers SimX1' *)
        

        (* Switch: '<S1>/Switch3' incorporates:
         *  Constant: '<S1>/Constant2' *)

        IF I_Cntr_Reset_On THEN 
            I_reset := DINT_TO_LREAL(rtb_I_Reset);
        ELSE 
            I_reset := 0.0;
        END_IF;

        (* End of Switch: '<S1>/Switch3' *)
        

        (* DiscreteIntegrator: '<S1>/Discrete-Time Integrator' *)

        IF I_reset <> 0.0 THEN 
            c_DiscreteTimeIntegrator_DS := 0.0;
        END_IF;

        (* SignalConversion: '<S4>/ConcatBufferAtVector ConcatenateIn1' *)
        VectorConcatenate[0] := k_AD_Num;
        (* Gain: '<S4>/Gain1' *)
        VectorConcatenate[1] :=  -k_AD_Num;
        (* DiscreteTransferFcn: '<S4>/Transfer Fcn1 1' incorporates:
         *  Gain: '<S4>/Cylinder Area Ratio'
         *  Sum: '<S4>/Load Pressure' *)
        TransferFcn11_tmp := (p_A - (0.710059171597633 * p_B)) - (-0.997 * TransferFcn11_states);
        u_AD := (VectorConcatenate[0] * TransferFcn11_tmp) + (VectorConcatenate[1] * TransferFcn11_states);
        (* Switch: '<S1>/Switch' incorporates:
         *  Constant: '<S1>/Constant'
         *  DiscreteIntegrator: '<S1>/Discrete-Time Integrator' *)

        IF I_Cntr_On THEN 
            u_I := c_DiscreteTimeIntegrator_DS;
        ELSE 
            u_I := 0.0;
        END_IF;

        (* End of Switch: '<S1>/Switch' *)
        

        (* Switch: '<S1>/Switch1' incorporates:
         *  Constant: '<S1>/Constant1'
         *  Sum: '<S1>/Sum5' *)

        IF FB_Cntr_On THEN 
            rtb_LoadPressure := u_P + u_I;
        ELSE 
            rtb_LoadPressure := 0.0;
        END_IF;

        (* End of Switch: '<S1>/Switch1' *)
        

        (* Saturate: '<S1>/Saturation1' *)

        IF rtb_LoadPressure >= 1.0 THEN 
            rtb_Saturation1 := 1.0;
        ELSIF rtb_LoadPressure > -1.0 THEN 
            rtb_Saturation1 := rtb_LoadPressure;
        ELSE 
            rtb_Saturation1 := -1.0;
        END_IF;

        (* End of Saturate: '<S1>/Saturation1' *)
        

        (* Switch: '<S1>/Switch4' incorporates:
         *  Constant: '<S1>/Constant3' *)

        IF  NOT Active_Damper_On THEN 
            u_AD := 0.0;
        END_IF;

        (* End of Switch: '<S1>/Switch4' *)
        

        (* Gain: '<S1>/Gain' incorporates:
         *  Sum: '<S1>/Sum6' *)
        rtb_Gain :=  -((u_FF + rtb_Saturation1) - u_AD);
        (* Saturate: '<S1>/Saturation5' *)

        IF rtb_Gain >= 1.0 THEN 
            rtb_Gain := 1.0;
        ELSIF  NOT (rtb_Gain > -1.0) THEN 
            rtb_Gain := -1.0;
        END_IF;

        (* End of Saturate: '<S1>/Saturation5' *)
        

        (* MATLAB Function: '<S1>/Anti DB From Jespers SimX' *)
        (* MATLAB Function 'VCC_Controller_FF_PI_AD1/Anti DB From Jespers SimX': '<S2>:1' *)
        (* '<S2>:1:5' u_DCV = 0; *)
        (* '<S2>:1:7' if (I_Reset == 1) &amp;&amp; (Tuning_Mode == 0) *)

        IF (rtb_I_Reset = 1) AND ( NOT Tuning_Mode_On) THEN 
            (* Outport: '<Root>/u_DCV' *)
            (* '<S2>:1:8' u_DCV = 0; *)
            u_DCV := 0.0;
        ELSIF rtb_Gain < -0.001 THEN 
            (* Outport: '<Root>/u_DCV' *)
            (* '<S2>:1:9' elseif (u_DCV_ref < -0.001) *)
            (* '<S2>:1:10' u_DCV = -DB_Up + (1-DB_Up)*u_DCV_ref; *)
            u_DCV := ((1.0 - DB_Up) * rtb_Gain) + ( -DB_Up);
        ELSIF rtb_Gain > 0.001 THEN 
            (* Outport: '<Root>/u_DCV' *)
            (* '<S2>:1:11' elseif (u_DCV_ref > 0.001) *)
            (* '<S2>:1:12' u_DCV = DB_Down + (1-DB_Down)*u_DCV_ref; *)
            u_DCV := ((1.0 - DB_Down) * rtb_Gain) + DB_Down;
        ELSE 
            (* Outport: '<Root>/u_DCV' *)
            (* '<S2>:1:13' else *)
            (* '<S2>:1:14' u_DCV = 0; *)
            u_DCV := 0.0;
        END_IF;

        (* End of MATLAB Function: '<S1>/Anti DB From Jespers SimX' *)
        

        (* Update for DiscreteIntegrator: '<S1>/Discrete-Time Integrator' incorporates:
         *  Product: '<S1>/Divide'
         *  Product: '<S1>/Product2'
         *  Sum: '<S1>/Sum2'
         *  Sum: '<S1>/Sum3' *)
        c_DiscreteTimeIntegrator_DS := (((((rtb_Saturation1 - rtb_LoadPressure) / k_P) + Pos_Error) * k_I) * 0.001) + c_DiscreteTimeIntegrator_DS;
        (* Update for DiscreteTransferFcn: '<S4>/Transfer Fcn1 1' *)
        TransferFcn11_states := TransferFcn11_tmp;
END_CASE;

END_FUNCTION_BLOCK

// IndraMotionMlc1/Application/VCC_SP_Ramp_Generator
FUNCTION_BLOCK VCC_SP_Ramp_Generator
VAR_INPUT
	Enable: BOOL;
	x0: LREAL;
	v0: LREAL;
	Position_SP: LREAL;
	Velocity_SP: LREAL;
	t0: LREAL;
	t_Ramp: LREAL;
	t_Hold_Pos: LREAL;
	CyclicTime: LREAL;
END_VAR
VAR_OUTPUT
	Position_Ref: LREAL;
	Velocity_Ref: LREAL;
	T: LREAL;
	Error: LREAL;
END_VAR
VAR
	Error_0: DINT;
	tHold_Up_Up_Up: LREAL;
	x1: LREAL;
	x4: LREAL;
	rtb_Saturation3: LREAL;
	a_tmp: LREAL;
	a_tmp_tmp: LREAL;
	a_tmp_0: LREAL;
	a_tmp_tmp_0: LREAL;
	a_tmp_tmp_1: LREAL;
	a_tmp_tmp_2: LREAL;
	x4_tmp: LREAL;
	x1_tmp: LREAL;
END_VAR


(* Saturate: '<S1>/Saturation3' *)

IF Position_SP >= 500.0 THEN 
    rtb_Saturation3 := 500.0;
ELSIF Position_SP > 0.0 THEN 
    rtb_Saturation3 := Position_SP;
ELSE 
    rtb_Saturation3 := 0.0;
END_IF;

(* End of Saturate: '<S1>/Saturation3' *)


(* Saturate: '<S1>/Saturation2' *)

IF Velocity_SP >= 150.0 THEN 
    Position_Ref := 150.0;
ELSIF Velocity_SP > 0.0 THEN 
    Position_Ref := Velocity_SP;
ELSE 
    Position_Ref := 0.0;
END_IF;

(* End of Saturate: '<S1>/Saturation2' *)


(* MATLAB Function: '<S1>/WaveSignal' *)
(* MATLAB Function 'Ramp_Test1/WaveSignal': '<S2>:1' *)
(* '<S2>:1:2' x_SP = x_ref - x0; *)
(* '<S2>:1:3' vs=v_ref; *)
(* '<S2>:1:4' slopeExt=v0-vs; *)
(* '<S2>:1:5' slopeRetr=-vs-v0; *)
(* '<S2>:1:7' as = vs/tRamp; *)
(* '<S2>:1:8' s_acc=(vs^2-v0^2)/as; *)
(* '<S2>:1:10' tHold_Up_Up_Up=(x_SP-s_acc)/vs; *)
tHold_Up_Up_Up := ((rtb_Saturation3 - x0) - (((Position_Ref * Position_Ref) - (v0 * v0)) / (Position_Ref / t_Ramp))) / Position_Ref;
(* '<S2>:1:12' if tHold_Up_Up_Up < 0 *)

IF tHold_Up_Up_Up < 0.0 THEN 
    (* '<S2>:1:13' Error = 1; *)
    Error_0 := 1;
ELSE 
    (* '<S2>:1:14' else *)
    (* '<S2>:1:15' Error = 0; *)
    Error_0 := 0;
END_IF;

(* '<S2>:1:18' t1=tRamp; *)
(* '<S2>:1:19' t2=tHold_Up_Up_Up; *)
(* '<S2>:1:20' t3=tRamp; *)
(* '<S2>:1:21' t4=tWait; *)
(* '<S2>:1:22' t5=t1; *)
(* '<S2>:1:23' t6=t2; *)
(* '<S2>:1:24' t7=t3; *)
(* '<S2>:1:26' x = x0; *)
(* '<S2>:1:27' x1 = x0 + v0*((t0+t1)-t0)-(slopeExt/t1)*((t0+t1)-t0)^2/2; *)
a_tmp_tmp := t0 + t_Ramp;
a_tmp := a_tmp_tmp - t0;
x1_tmp := (v0 - Position_Ref) / t_Ramp;
x1 := ((a_tmp * v0) + x0) - ((x1_tmp * (a_tmp * a_tmp)) / 2.0);
(* '<S2>:1:28' x2 = x1 + vs*((t0+t1+t2)-(t0+t1)); *)
(* '<S2>:1:29' x4 = x_ref - v0*((t0+t1+t2+t3+t4+t5)-(t0+t1+t2+t3+t4))+(slopeRetr/t5)*((t0+t1+t2+t3+t4+t5)-(t0+t1+t2+t3+t4))^2/2; *)
a_tmp_tmp_0 := a_tmp_tmp + tHold_Up_Up_Up;
a_tmp_tmp_1 := a_tmp_tmp_0 + t_Ramp;
a_tmp := a_tmp_tmp_1 + t_Hold_Pos;
a_tmp_tmp_2 := a_tmp + t_Ramp;
a_tmp_0 := a_tmp_tmp_2 - a_tmp;
x4_tmp := (( -Position_Ref) - v0) / t_Ramp;
x4 := (rtb_Saturation3 - (a_tmp_0 * v0)) + ((x4_tmp * (a_tmp_0 * a_tmp_0)) / 2.0);
(* '<S2>:1:30' x5 = x4-vs*((t0+t1+t2+t3+t4+t5+t6)-(t0+t1+t2+t3+t4+t5)); *)
(* '<S2>:1:32' if Error == 1 *)

IF Error_0 = 1 THEN 
    (* '<S2>:1:33' x = x0; *)
    rtb_Saturation3 := x0;
    (* '<S2>:1:34' v = v0; *)
    Position_Ref := v0;
ELSIF (CyclicTime >= 0.0) AND (CyclicTime < t0) THEN 
    (* '<S2>:1:35' elseif t>=0 &amp;&amp; t<t0 *)
    (* '<S2>:1:36' x = x0; *)
    rtb_Saturation3 := x0;
    (* '<S2>:1:37' v = v0; *)
    Position_Ref := v0;
ELSIF (CyclicTime >= t0) AND (CyclicTime < a_tmp_tmp) THEN 
    (* '<S2>:1:38' elseif t>=t0 &amp;&amp; t<(t0+t1) *)
    (* '<S2>:1:39' x = x0 + v0*(t-t0)-(slopeExt/t1)*(t-t0)^2/2; *)
    a_tmp := CyclicTime - t0;
    rtb_Saturation3 := ((a_tmp * v0) + x0) - ((x1_tmp * (a_tmp * a_tmp)) / 2.0);
    (* '<S2>:1:40' v = v0-(slopeExt/t1)*(t-t0); *)
    Position_Ref := v0 - (x1_tmp * a_tmp);
ELSIF (CyclicTime >= a_tmp_tmp) AND (CyclicTime < a_tmp_tmp_0) THEN 
    (* '<S2>:1:41' elseif t>=(t0+t1) &amp;&amp; t<(t0+t1+t2) *)
    (* '<S2>:1:42' x = x1 + vs*(t-(t0+t1)); *)
    rtb_Saturation3 := ((CyclicTime - a_tmp_tmp) * Position_Ref) + x1;
    (* '<S2>:1:43' v = vs; *)
ELSIF (CyclicTime >= a_tmp_tmp_0) AND (CyclicTime < a_tmp_tmp_1) THEN 
    (* '<S2>:1:44' elseif t>=(t0+t1+t2) &amp;&amp; t<(t0+t1+t2+t3) *)
    (* '<S2>:1:45' x = x2+vs*(t-(t0+t1+t2))+(slopeExt/t3)*(t-(t0+t1+t2))^2/2; *)
    a_tmp := CyclicTime - a_tmp_tmp_0;
    rtb_Saturation3 := ((((a_tmp_tmp_0 - a_tmp_tmp) * Position_Ref) + x1) + (a_tmp * Position_Ref)) + ((x1_tmp * (a_tmp * a_tmp)) / 2.0);
    (* '<S2>:1:46' v = vs+(slopeExt/t3)*(t-(t0+t1+t2)); *)
    Position_Ref := (a_tmp * x1_tmp) + Position_Ref;
ELSIF (CyclicTime >= a_tmp_tmp_1) AND (CyclicTime < a_tmp) THEN 
    (* '<S2>:1:47' elseif t>=(t0+t1+t2+t3) &amp;&amp; t<(t0+t1+t2+t3+t4) *)
    (* '<S2>:1:48' x = x_ref; *)
    (* '<S2>:1:49' v = v0; *)
    Position_Ref := v0;
ELSIF (CyclicTime >= a_tmp) AND (CyclicTime < a_tmp_tmp_2) THEN 
    (* '<S2>:1:50' elseif t>=(t0+t1+t2+t3+t4) &amp;&amp; t<(t0+t1+t2+t3+t4+t5) *)
    (* '<S2>:1:51' x = x_ref - v0*(t-(t0+t1+t2+t3+t4))+(slopeRetr/t5)*(t-(t0+t1+t2+t3+t4))^2/2; *)
    a_tmp := CyclicTime - a_tmp;
    rtb_Saturation3 := (rtb_Saturation3 - (a_tmp * v0)) + ((x4_tmp * (a_tmp * a_tmp)) / 2.0);
    (* '<S2>:1:52' v = v0+(slopeRetr/t5)*(t-(t0+t1+t2+t3+t4)); *)
    Position_Ref := (a_tmp * x4_tmp) + v0;
ELSE 
    rtb_Saturation3 := a_tmp_tmp_2 + tHold_Up_Up_Up;

    IF (CyclicTime >= a_tmp_tmp_2) AND (CyclicTime < rtb_Saturation3) THEN 
        (* '<S2>:1:53' elseif t>=(t0+t1+t2+t3+t4+t5) &amp;&amp; t<(t0+t1+t2+t3+t4+t5+t6) *)
        (* '<S2>:1:54' x = x4-vs*(t-(t0+t1+t2+t3+t4+t5)); *)
        rtb_Saturation3 := x4 - ((CyclicTime - a_tmp_tmp_2) * Position_Ref);
        (* '<S2>:1:55' v = -vs; *)
        Position_Ref :=  -Position_Ref;
    ELSIF (CyclicTime >= rtb_Saturation3) AND (CyclicTime < (rtb_Saturation3 + t_Ramp)) THEN 
        (* '<S2>:1:56' elseif t>=(t0+t1+t2+t3+t4+t5+t6) &amp;&amp; t<(t0+t1+t2+t3+t4+t5+t6+t7) *)
        (* '<S2>:1:57' x = x5-vs*(t-(t0+t1+t2+t3+t4+t5+t6))-(slopeRetr/t3)*(t-(t0+t1+t2+t3+t4+t5+t6))^2/2; *)
        a_tmp := CyclicTime - rtb_Saturation3;
        rtb_Saturation3 := ((x4 - ((rtb_Saturation3 - a_tmp_tmp_2) * Position_Ref)) - (a_tmp * Position_Ref)) - ((x4_tmp * (a_tmp * a_tmp)) / 2.0);
        (* '<S2>:1:58' v = -vs-(slopeRetr/t3)*(t-(t0+t1+t2+t3+t4+t5+t6)); *)
        Position_Ref := ( -Position_Ref) - (a_tmp * x4_tmp);
    ELSE 
        (* '<S2>:1:59' else *)
        (* '<S2>:1:60' x = x0; *)
        rtb_Saturation3 := x0;
        (* '<S2>:1:61' v = v0; *)
        Position_Ref := v0;
    END_IF;

END_IF;

(* Switch: '<S1>/Switch' *)
(* '<S2>:1:64' T = t0+t1+t2+t3+t4+t5+t6+t7; *)

IF  NOT Enable THEN 
    Position_Ref := v0;
END_IF;

(* End of Switch: '<S1>/Switch' *)


(* Saturate: '<S1>/Saturation' *)

IF Position_Ref >= 150.0 THEN 
    (* Outport: '<Root>/Velocity_Ref' *)
    Velocity_Ref := 150.0;
ELSIF Position_Ref > -150.0 THEN 
    (* Outport: '<Root>/Velocity_Ref' *)
    Velocity_Ref := Position_Ref;
ELSE 
    (* Outport: '<Root>/Velocity_Ref' *)
    Velocity_Ref := -150.0;
END_IF;

(* End of Saturate: '<S1>/Saturation' *)


(* Switch: '<S1>/Switch1' *)

IF Enable THEN 
    Position_Ref := rtb_Saturation3;
ELSE 
    Position_Ref := x0;
END_IF;

(* End of Switch: '<S1>/Switch1' *)


(* Saturate: '<S1>/Saturation1' *)

IF Position_Ref >= 500.0 THEN 
    (* Outport: '<Root>/Position_Ref' *)
    Position_Ref := 500.0;
ELSIF  NOT (Position_Ref > 0.0) THEN 
    (* Outport: '<Root>/Position_Ref' *)
    Position_Ref := 0.0;
END_IF;

(* End of Saturate: '<S1>/Saturation1' *)


(* Outport: '<Root>/T' incorporates:
 *  MATLAB Function: '<S1>/WaveSignal' *)
T := ((((((t0 + t_Ramp) + tHold_Up_Up_Up) + t_Ramp) + t_Hold_Pos) + t_Ramp) + tHold_Up_Up_Up) + t_Ramp;
(* Outport: '<Root>/Error' incorporates:
 *  MATLAB Function: '<S1>/WaveSignal' *)
Error := DINT_TO_LREAL(Error_0);

END_FUNCTION_BLOCK

// IndraMotionMlc1/Application/VCC_Controller_PI_FF
FUNCTION_BLOCK VCC_Controller_PI_FF
VAR_INPUT
	ssMethodType: SINT;
	FB_Cntr_On: BOOL;
	I_Cntr_On: BOOL;
	I_Cntr_Reset_On: BOOL;
	Qmax: LREAL;
	Clock: LREAL;
	k_P: LREAL;
	k_I: LREAL;
	Pos_Ref: LREAL;
	Vel_Ref: LREAL;
	Pos_FB: LREAL;
END_VAR
VAR_OUTPUT
	Pos_Error: LREAL;
	u_P: LREAL;
	u_I: LREAL;
	I_reset: LREAL;
	uV: LREAL;
	uFF: LREAL;
END_VAR
VAR
	rtb_Saturation1: LREAL;
	rtb_Sum3: LREAL;
	rtb_Saturation2: LREAL;
	c_DiscreteTimeIntegrator_DS: LREAL;
END_VAR



CASE ssMethodType OF
    0: 
        (* InitializeConditions for DiscreteIntegrator: '<S1>/Discrete-Time Integrator' *)
        c_DiscreteTimeIntegrator_DS := 0.0;
    1: 
        (* MATLAB Function: '<S1>/Controller_Reset' *)
        (* MATLAB Function 'VCC_Controller_PI_FF/Controller_Reset': '<S2>:1' *)
        (* '<S2>:1:3' I_Reset = 1; *)
        (* '<S2>:1:5' if Clock > 0 *)

        IF Clock > 0.0 THEN 
            (* '<S2>:1:6' I_Reset = 0; *)
            I_reset := 0.0;
        ELSE 
            (* '<S2>:1:7' else *)
            (* '<S2>:1:8' I_Reset = 1; *)
            I_reset := 1.0;
        END_IF;

        (* End of MATLAB Function: '<S1>/Controller_Reset' *)
        

        (* Switch: '<S1>/Switch3' incorporates:
         *  Constant: '<S1>/Constant2' *)

        IF  NOT I_Cntr_Reset_On THEN 
            I_reset := 0.0;
        END_IF;

        (* End of Switch: '<S1>/Switch3' *)
        

        (* DiscreteIntegrator: '<S1>/Discrete-Time Integrator' *)

        IF I_reset <> 0.0 THEN 
            c_DiscreteTimeIntegrator_DS := 0.0;
        END_IF;

        (* Sum: '<S1>/Sum1' *)
        Pos_Error := Pos_Ref - Pos_FB;
        (* Product: '<S1>/Product' *)
        u_P := k_P * Pos_Error;
        (* Switch: '<S1>/Switch' incorporates:
         *  Constant: '<S1>/Constant'
         *  DiscreteIntegrator: '<S1>/Discrete-Time Integrator' *)

        IF I_Cntr_On THEN 
            u_I := c_DiscreteTimeIntegrator_DS;
        ELSE 
            u_I := 0.0;
        END_IF;

        (* End of Switch: '<S1>/Switch' *)
        

        (* Switch: '<S1>/Switch1' incorporates:
         *  Constant: '<S1>/Constant1'
         *  Sum: '<S1>/Sum5' *)

        IF FB_Cntr_On THEN 
            uFF := u_P + u_I;
        ELSE 
            uFF := 0.0;
        END_IF;

        (* End of Switch: '<S1>/Switch1' *)
        

        (* Saturate: '<S1>/Saturation1' *)

        IF uFF >= 1.0 THEN 
            rtb_Saturation1 := 1.0;
        ELSIF uFF > -1.0 THEN 
            rtb_Saturation1 := uFF;
        ELSE 
            rtb_Saturation1 := -1.0;
        END_IF;

        (* End of Saturate: '<S1>/Saturation1' *)
        

        (* Sum: '<S1>/Sum3' *)
        rtb_Sum3 := rtb_Saturation1 - uFF;
        (* Switch: '<S1>/Switch2' incorporates:
         *  Constant: '<S1>/Annnulus_Area'
         *  Constant: '<S1>/Bore_Area'
         *  Product: '<S1>/Product1'
         *  Product: '<S1>/Product3' *)

        IF Vel_Ref >= 0.0 THEN 
            uFF := 3318.3 * Vel_Ref;
        ELSE 
            uFF := Vel_Ref * 2356.2;
        END_IF;

        (* End of Switch: '<S1>/Switch2' *)
        

        (* Product: '<S1>/Divide2' incorporates:
         *  Gain: '<S1>/Gain1'
         *  Gain: '<S1>/Gain2' *)
        uFF := ((1.0E-9 * uFF) * 60000.0) / Qmax;
        (* Saturate: '<S1>/Saturation2' *)

        IF uFF >= 1.0 THEN 
            rtb_Saturation2 := 1.0;
        ELSIF uFF > -1.0 THEN 
            rtb_Saturation2 := uFF;
        ELSE 
            rtb_Saturation2 := -1.0;
        END_IF;

        (* End of Saturate: '<S1>/Saturation2' *)
        

        (* Outport: '<Root>/uV' incorporates:
         *  Sum: '<S1>/Sum6' *)
        uV := rtb_Saturation2 + rtb_Saturation1;
        (* Update for DiscreteIntegrator: '<S1>/Discrete-Time Integrator' incorporates:
         *  Product: '<S1>/Divide'
         *  Product: '<S1>/Product2'
         *  Sum: '<S1>/Sum2' *)
        c_DiscreteTimeIntegrator_DS := ((((rtb_Sum3 / k_P) + Pos_Error) * k_I) * 0.001) + c_DiscreteTimeIntegrator_DS;
END_CASE;

END_FUNCTION_BLOCK

// IndraMotionMlc1/Application/VCC_PRV_Control
PROGRAM VCC_PRV_Control
VAR_INPUT
	 Enable: BOOL;
END_VAR
VAR_OUTPUT
	
END_VAR


VAR
	VCC_PRV_Mapping_0: VCC_PRV_Mapping;
	PRV_Pressure_SP_Opening: WORD;
	PRV_Valve_Opening: WORD;
	Discrete_Lowpass_Filter0_0: Discrete_Lowpass_Filter0;
	VCC_PV_Controller_0: VCC_PV_Controller;
	u_PV: WORD;
	u_PRV: LREAL;
	p_C_ref: LREAL;
	k_P: LREAL;
	k_I: LREAL;
END_VAR
VAR // added by the converter: edge detectors and wires of the graphical bodies
    _w1, _w2, _w3 : BOOL;
END_VAR

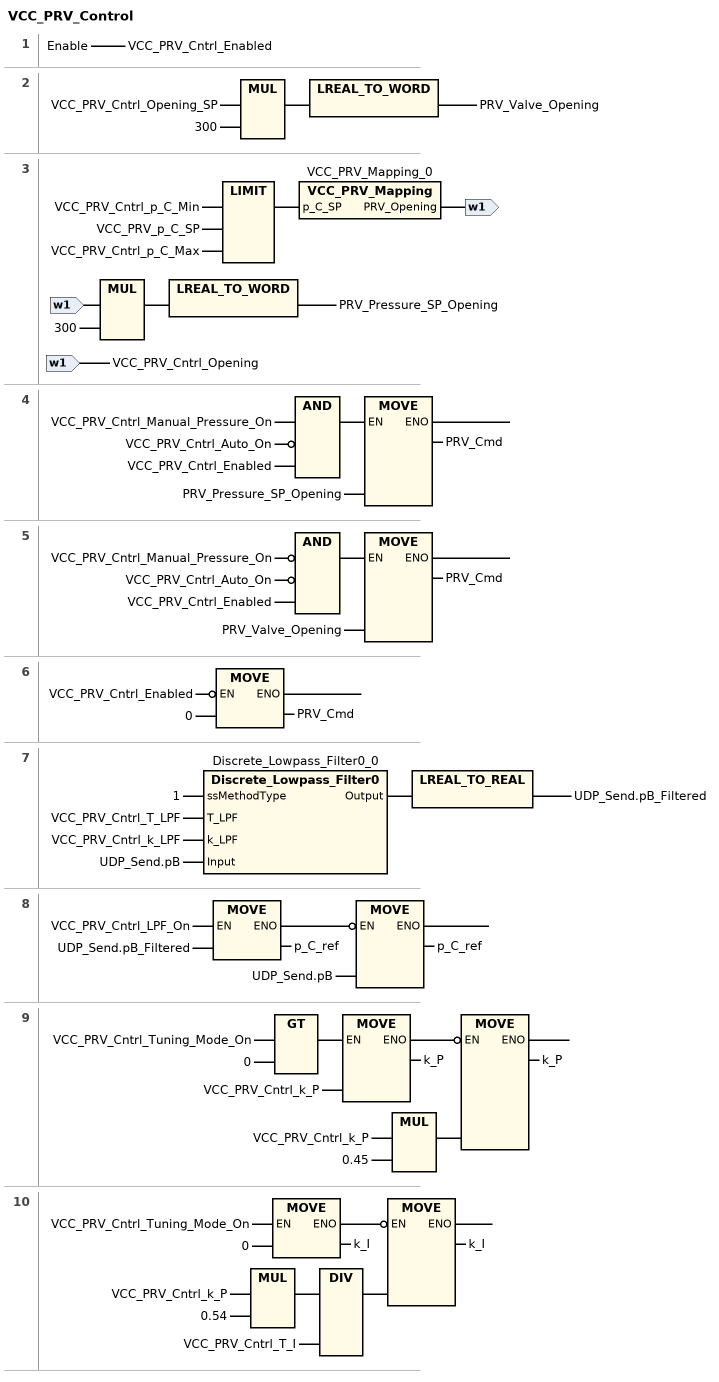
// NETWORK 1
VCC_PRV_Cntrl_Enabled := Enable;

// NETWORK 2
PRV_Valve_Opening := LREAL_TO_WORD(VCC_PRV_Cntrl_Opening_SP * 300);

// NETWORK 3
VCC_PRV_Mapping_0(p_C_SP := LIMIT(VCC_PRV_Cntrl_p_C_Min, VCC_PRV_p_C_SP, VCC_PRV_Cntrl_p_C_Max)); // VCC_PRV_Mapping
PRV_Pressure_SP_Opening := LREAL_TO_WORD(VCC_PRV_Mapping_0.PRV_Opening * 300);
VCC_PRV_Cntrl_Opening := VCC_PRV_Mapping_0.PRV_Opening;

// NETWORK 4
IF VCC_PRV_Cntrl_Manual_Pressure_On AND NOT VCC_PRV_Cntrl_Auto_On AND VCC_PRV_Cntrl_Enabled THEN
    PRV_Cmd := PRV_Pressure_SP_Opening;
END_IF

// NETWORK 5
IF NOT VCC_PRV_Cntrl_Manual_Pressure_On AND NOT VCC_PRV_Cntrl_Auto_On AND VCC_PRV_Cntrl_Enabled THEN
    PRV_Cmd := PRV_Valve_Opening;
END_IF

// NETWORK 6
IF NOT VCC_PRV_Cntrl_Enabled THEN PRV_Cmd := 0; END_IF

// NETWORK 7
Discrete_Lowpass_Filter0_0(
    ssMethodType := 1,
    T_LPF := VCC_PRV_Cntrl_T_LPF,
    k_LPF := VCC_PRV_Cntrl_k_LPF,
    Input := UDP_Send.pB); // Discrete_Lowpass_Filter0
UDP_Send.pB_Filtered := LREAL_TO_REAL(Discrete_Lowpass_Filter0_0.Output);

// NETWORK 8
_w1 := VCC_PRV_Cntrl_LPF_On;
IF _w1 THEN p_C_ref := UDP_Send.pB_Filtered; END_IF
IF NOT _w1 THEN p_C_ref := UDP_Send.pB; END_IF

// NETWORK 9
_w2 := VCC_PRV_Cntrl_Tuning_Mode_On > 0;
IF _w2 THEN k_P := VCC_PRV_Cntrl_k_P; END_IF
IF NOT _w2 THEN k_P := VCC_PRV_Cntrl_k_P * 0.45; END_IF

// NETWORK 10
_w3 := VCC_PRV_Cntrl_Tuning_Mode_On;
IF _w3 THEN k_I := 0; END_IF
IF NOT _w3 THEN k_I := (VCC_PRV_Cntrl_k_P * 0.54) / VCC_PRV_Cntrl_T_I; END_IF

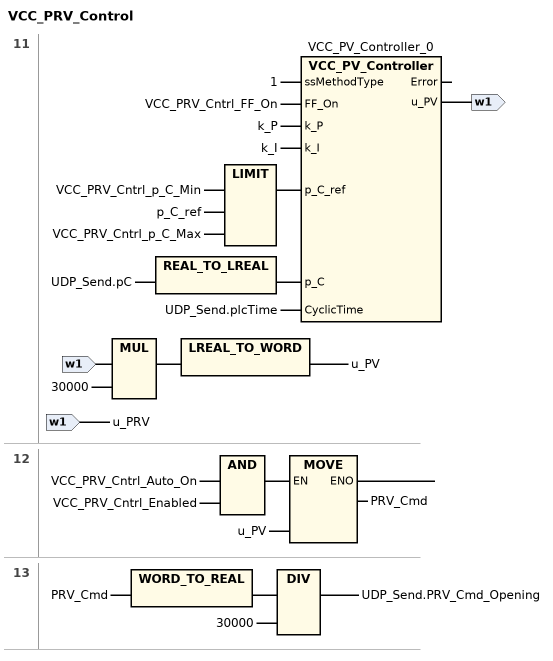
// NETWORK 11
VCC_PV_Controller_0(
    ssMethodType := 1,
    FF_On := VCC_PRV_Cntrl_FF_On,
    k_P := k_P,
    k_I := k_I,
    p_C_ref := LIMIT(VCC_PRV_Cntrl_p_C_Min, p_C_ref, VCC_PRV_Cntrl_p_C_Max),
    p_C := REAL_TO_LREAL(UDP_Send.pC),
    CyclicTime := UDP_Send.plcTime); // VCC_PV_Controller
u_PV := LREAL_TO_WORD(VCC_PV_Controller_0.u_PV * 30000);
u_PRV := VCC_PV_Controller_0.u_PV;

// NETWORK 12
IF VCC_PRV_Cntrl_Auto_On AND VCC_PRV_Cntrl_Enabled THEN PRV_Cmd := u_PV; END_IF

// NETWORK 13
UDP_Send.PRV_Cmd_Opening := WORD_TO_REAL(PRV_Cmd) / 30000;

END_PROGRAM

// IndraMotionMlc1/Application/VCC_PRV_Mapping
FUNCTION_BLOCK VCC_PRV_Mapping
VAR_INPUT
	p_C_SP: LREAL;
END_VAR
VAR_OUTPUT
	PRV_Opening: LREAL;
END_VAR
VAR
	frac: LREAL;
	iRght: UDINT;
	iLeft: UDINT;
	bpIdx: UDINT;
	uvsQ_tableData: ARRAY[0..16] OF LREAL := [0.0, 5.0, 10.0, 15.0, 20.0, 25.0, 30.0, 35.0, 40.0, 45.0, 50.0, 55.0, 60.0, 65.0, 70.0, 75.0, 100.0];
	uvsQ_bp01Data: ARRAY[0..16] OF LREAL := [0.0, 3.0, 16.0, 31.0, 48.0, 61.0, 74.0, 87.0, 100.0, 114.0, 128.0, 142.0, 155.0, 168.0, 174.0, 181.0, 182.0];
END_VAR


(* Lookup_n-D: '<S1>/ u vs Q ' *)
(* Lookup 1-D
   Search method: 'binary'
   Use previous index: 'off'
   Interpolation method: 'Linear'
   Extrapolation method: 'Linear'
   Use last breakpoint for index at or above upper limit: 'off'
   Remove protection against out-of-range input in generated code: 'off' *)
(* Prelookup - Index and Fraction
   Index Search method: 'binary'
   Extrapolation method: 'Linear'
   Use previous index: 'off'
   Use last breakpoint for index at or above upper limit: 'off'
   Remove protection against out-of-range input in generated code: 'off' *)

IF p_C_SP <= 0.0 THEN 
    iLeft := 0;
    frac := p_C_SP / 3.0;
ELSIF p_C_SP < 182.0 THEN 
    (* Binary Search *)
    bpIdx := 8;
    iLeft := 0;
    iRght := 16;
    WHILE (iRght - iLeft) > 1 DO

        IF p_C_SP < uvsQ_bp01Data[bpIdx] THEN 
            iRght := bpIdx;
        ELSE 
            iLeft := bpIdx;
        END_IF;

        bpIdx := DWORD_TO_UDINT(SHR(UDINT_TO_DWORD(iRght + iLeft), 1));
    END_WHILE;
    frac := (p_C_SP - uvsQ_bp01Data[iLeft]) / (uvsQ_bp01Data[iLeft + 1] - uvsQ_bp01Data[iLeft]);
ELSE 
    iLeft := 15;
    frac := p_C_SP - 181.0;
END_IF;

(* Outport: '<Root>/PRV_Opening' incorporates:
 *  Lookup_n-D: '<S1>/ u vs Q ' *)
(* Interpolation 1-D
   Interpolation method: 'Linear'
   Use last breakpoint for index at or above upper limit: 'off'
   Overflow mode: 'wrapping' *)
PRV_Opening := ((uvsQ_tableData[iLeft + 1] - uvsQ_tableData[iLeft]) * frac) + uvsQ_tableData[iLeft];

END_FUNCTION_BLOCK

// IndraMotionMlc1/Application/Discrete_Lowpass_Filter0
FUNCTION_BLOCK Discrete_Lowpass_Filter0
VAR_INPUT
	ssMethodType: SINT;
	T_LPF: LREAL;
	k_LPF: LREAL;
	Input: LREAL;
END_VAR
VAR_OUTPUT
	Output: LREAL;
END_VAR
VAR
	maxV: LREAL;
	rtb_Compare: BOOL;
	rtb_Product: LREAL;
	Integrator_PrevResetState: SINT;
	Integrator_IC_LOADING: USINT;
	Integrator_DSTATE: LREAL;
	Probe: ARRAY[0..1] OF LREAL;
END_VAR



CASE ssMethodType OF
    0: 
        (* Start for Probe: '<S1>/Probe' *)
        Probe[0] := 0.001;
        Probe[1] := 0.0;
        (* InitializeConditions for DiscreteIntegrator: '<S5>/Integrator' *)
        Integrator_IC_LOADING := 1;
        Integrator_PrevResetState := 0;
    1: 
        (* RelationalOperator: '<S2>/Compare' incorporates:
         *  Constant: '<S2>/Constant'
         *  Sum: '<S1>/Sum2' *)
        rtb_Compare := (T_LPF - Probe[0]) <= 0.0;
        (* Product: '<S1>/Product' *)
        rtb_Product := k_LPF * Input;
        (* DiscreteIntegrator: '<S5>/Integrator' *)

        IF Integrator_IC_LOADING <> 0 THEN 
            Integrator_DSTATE := rtb_Product;

            IF Integrator_DSTATE >= 210.0 THEN 
                Integrator_DSTATE := 210.0;
            ELSIF Integrator_DSTATE <= 0.0 THEN 
                Integrator_DSTATE := 0.0;
            END_IF;

        END_IF;


        IF rtb_Compare OR (Integrator_PrevResetState <> 0) THEN 
            Integrator_DSTATE := rtb_Product;

            IF Integrator_DSTATE >= 210.0 THEN 
                Integrator_DSTATE := 210.0;
            ELSIF Integrator_DSTATE <= 0.0 THEN 
                Integrator_DSTATE := 0.0;
            END_IF;

        END_IF;


        IF Integrator_DSTATE >= 210.0 THEN 
            Integrator_DSTATE := 210.0;
        ELSIF Integrator_DSTATE <= 0.0 THEN 
            Integrator_DSTATE := 0.0;
        END_IF;

        (* MinMax: '<S1>/Max' *)
        maxV := MAX(Probe[0], T_LPF);
        (* Outport: '<Root>/Output' incorporates:
         *  DiscreteIntegrator: '<S5>/Integrator' *)
        Output := Integrator_DSTATE;
        (* Update for DiscreteIntegrator: '<S5>/Integrator' incorporates:
         *  Fcn: '<S1>/Avoid Divide by Zero'
         *  MinMax: '<S1>/Max'
         *  Product: '<S1>/1//T'
         *  Sum: '<S1>/Sum1' *)
        Integrator_IC_LOADING := 0;
        Integrator_DSTATE := (((1.0 / ((BOOL_TO_LREAL(maxV = 0.0) * 2.2204460492503131E-16) + maxV)) * (rtb_Product - Integrator_DSTATE)) * 0.001) + Integrator_DSTATE;

        IF Integrator_DSTATE >= 210.0 THEN 
            Integrator_DSTATE := 210.0;
        ELSIF Integrator_DSTATE <= 0.0 THEN 
            Integrator_DSTATE := 0.0;
        END_IF;


        IF rtb_Compare THEN 
            Integrator_PrevResetState := 1;
        ELSE 
            Integrator_PrevResetState := 0;
        END_IF;

        (* End of Update for DiscreteIntegrator: '<S5>/Integrator' *)
END_CASE;

END_FUNCTION_BLOCK

// IndraMotionMlc1/Application/VCC_PV_Controller
FUNCTION_BLOCK VCC_PV_Controller
VAR_INPUT
	ssMethodType: SINT;
	FF_On: BOOL;
	k_P: LREAL;
	k_I: LREAL;
	p_C_ref: LREAL;
	p_C: LREAL;
	CyclicTime: LREAL;
END_VAR
VAR_OUTPUT
	Error: LREAL;
	u_PV: LREAL;
END_VAR
VAR
	frac: LREAL;
	iRght: UDINT;
	iLeft: UDINT;
	bpIdx: UDINT;
	rtb_Switch1: LREAL;
	rtb_Sum3: LREAL;
	c_DiscreteTimeIntegrator_DS: LREAL;
	pvsu_tableData: ARRAY[0..16] OF LREAL := [0.0, 0.05, 0.1, 0.15, 0.2, 0.25, 0.3, 0.35, 0.4, 0.45, 0.5, 0.55, 0.6, 0.65, 0.7, 0.75, 1.0];
	pvsu_bp01Data: ARRAY[0..16] OF LREAL := [0.0, 3.0, 16.0, 31.0, 48.0, 61.0, 74.0, 87.0, 100.0, 114.0, 128.0, 142.0, 155.0, 168.0, 174.0, 181.0, 182.0];
END_VAR



CASE ssMethodType OF
    0: 
        (* InitializeConditions for DiscreteIntegrator: '<S1>/Discrete-Time Integrator' *)
        c_DiscreteTimeIntegrator_DS := 0.0;
    1: 
        (* Switch: '<S1>/Switch1' incorporates:
         *  Constant: '<S1>/Constant1'
         *  Constant: '<S1>/Constant2' *)

        IF CyclicTime > 0.0 THEN 
            rtb_Switch1 := 0.0;
        ELSE 
            rtb_Switch1 := 1.0;
        END_IF;

        (* End of Switch: '<S1>/Switch1' *)
        

        (* DiscreteIntegrator: '<S1>/Discrete-Time Integrator' *)

        IF rtb_Switch1 <> 0.0 THEN 
            c_DiscreteTimeIntegrator_DS := 0.0;
        END_IF;

        (* Sum: '<S1>/Sum1' *)
        Error := p_C_ref - p_C;
        (* Sum: '<S1>/Sum5' incorporates:
         *  DiscreteIntegrator: '<S1>/Discrete-Time Integrator'
         *  Product: '<S1>/Product' *)
        u_PV := (k_P * Error) + c_DiscreteTimeIntegrator_DS;
        (* Saturate: '<S1>/Saturation1' *)

        IF u_PV >= 1.0 THEN 
            rtb_Switch1 := 1.0;
        ELSIF u_PV > 0.0 THEN 
            rtb_Switch1 := u_PV;
        ELSE 
            rtb_Switch1 := 0.0;
        END_IF;

        (* End of Saturate: '<S1>/Saturation1' *)
        

        (* Sum: '<S1>/Sum3' *)
        rtb_Sum3 := rtb_Switch1 - u_PV;
        (* Outputs for Atomic SubSystem: '<S1>/Feed_Forward' *)
        (* Lookup_n-D: '<S2>/ p vs u ' *)
        (* Lookup 1-D
           Search method: 'binary'
           Use previous index: 'off'
           Interpolation method: 'Linear'
           Extrapolation method: 'Linear'
           Use last breakpoint for index at or above upper limit: 'off'
           Remove protection against out-of-range input in generated code: 'off' *)
        (* Prelookup - Index and Fraction
           Index Search method: 'binary'
           Extrapolation method: 'Linear'
           Use previous index: 'off'
           Use last breakpoint for index at or above upper limit: 'off'
           Remove protection against out-of-range input in generated code: 'off' *)

        IF p_C_ref <= 0.0 THEN 
            iLeft := 0;
            frac := p_C_ref / 3.0;
        ELSIF p_C_ref < 182.0 THEN 
            (* Binary Search *)
            bpIdx := 8;
            iLeft := 0;
            iRght := 16;
            WHILE (iRght - iLeft) > 1 DO

                IF p_C_ref < pvsu_bp01Data[bpIdx] THEN 
                    iRght := bpIdx;
                ELSE 
                    iLeft := bpIdx;
                END_IF;

                bpIdx := DWORD_TO_UDINT(SHR(UDINT_TO_DWORD(iRght + iLeft), 1));
            END_WHILE;
            frac := (p_C_ref - pvsu_bp01Data[iLeft]) / (pvsu_bp01Data[iLeft + 1] - pvsu_bp01Data[iLeft]);
        ELSE 
            iLeft := 15;
            frac := p_C_ref - 181.0;
        END_IF;

        (* End of Outputs for SubSystem: '<S1>/Feed_Forward' *)
        

        (* Switch: '<S1>/Switch' incorporates:
         *  Constant: '<S1>/Constant'
         *  Lookup_n-D: '<S2>/ p vs u ' *)
        (* Interpolation 1-D
           Interpolation method: 'Linear'
           Use last breakpoint for index at or above upper limit: 'off'
           Overflow mode: 'wrapping' *)

        IF FF_On THEN 
            (* Outputs for Atomic SubSystem: '<S1>/Feed_Forward' *)
            u_PV := ((pvsu_tableData[iLeft + 1] - pvsu_tableData[iLeft]) * frac) + pvsu_tableData[iLeft];
            (* End of Outputs for SubSystem: '<S1>/Feed_Forward' *)
        ELSE 
            u_PV := 0.0;
        END_IF;

        (* End of Switch: '<S1>/Switch' *)
        

        (* Sum: '<S1>/Sum4' *)
        u_PV := u_PV + rtb_Switch1;
        (* Saturate: '<S1>/Saturation2' *)

        IF u_PV >= 1.0 THEN 
            (* Outport: '<Root>/u_PV' *)
            u_PV := 1.0;
        ELSIF  NOT (u_PV > 0.0) THEN 
            (* Outport: '<Root>/u_PV' *)
            u_PV := 0.0;
        END_IF;

        (* End of Saturate: '<S1>/Saturation2' *)
        

        (* Update for DiscreteIntegrator: '<S1>/Discrete-Time Integrator' incorporates:
         *  Product: '<S1>/Divide'
         *  Product: '<S1>/Product2'
         *  Sum: '<S1>/Sum2' *)
        c_DiscreteTimeIntegrator_DS := ((((rtb_Sum3 / k_P) + Error) * k_I) * 0.001) + c_DiscreteTimeIntegrator_DS;
END_CASE;

END_FUNCTION_BLOCK

// IndraMotionMlc1/Application/HMI
PROGRAM HMI
VAR
	CyclSercosChnl_0: CyclSercosChnl;
	Real_Time_Counter_0: Real_Time_Counter;
	Input_Signals_0: Input_Signals;
END_VAR
VAR // added by the converter: edge detectors and wires of the graphical bodies
    _w1, _w2, _w3 : BOOL;
END_VAR

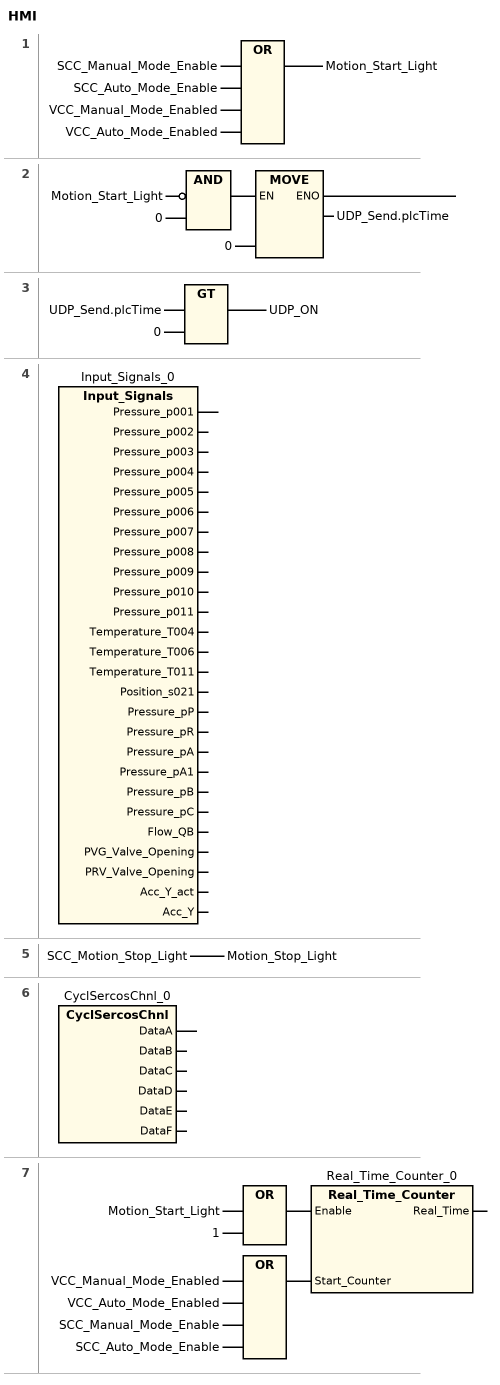
// NETWORK 1
Motion_Start_Light := SCC_Manual_Mode_Enable OR SCC_Auto_Mode_Enable OR VCC_Manual_Mode_Enabled OR VCC_Auto_Mode_Enabled;

// NETWORK 2
IF NOT Motion_Start_Light AND 0 THEN UDP_Send.plcTime := 0; END_IF

// NETWORK 3
UDP_ON := UDP_Send.plcTime > 0;

// NETWORK 4
Input_Signals_0(); // Input_Signals

// NETWORK 5
Motion_Stop_Light := SCC_Motion_Stop_Light;

// NETWORK 6
CyclSercosChnl_0(); // CyclSercosChnl

// NETWORK 7
Real_Time_Counter_0(Enable := Motion_Start_Light OR 1, Start_Counter := VCC_Manual_Mode_Enabled OR VCC_Auto_Mode_Enabled OR SCC_Manual_Mode_Enable OR SCC_Auto_Mode_Enable); // Real_Time_Counter

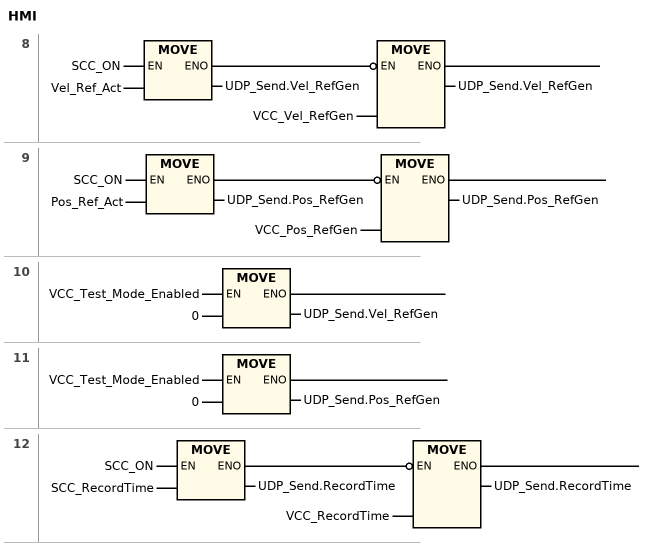
// NETWORK 8
_w1 := SCC_ON;
IF _w1 THEN UDP_Send.Vel_RefGen := Vel_Ref_Act; END_IF
IF NOT _w1 THEN UDP_Send.Vel_RefGen := VCC_Vel_RefGen; END_IF

// NETWORK 9
_w2 := SCC_ON;
IF _w2 THEN UDP_Send.Pos_RefGen := Pos_Ref_Act; END_IF
IF NOT _w2 THEN UDP_Send.Pos_RefGen := VCC_Pos_RefGen; END_IF

// NETWORK 10
IF VCC_Test_Mode_Enabled THEN UDP_Send.Vel_RefGen := 0; END_IF

// NETWORK 11
IF VCC_Test_Mode_Enabled THEN UDP_Send.Pos_RefGen := 0; END_IF

// NETWORK 12
_w3 := SCC_ON;
IF _w3 THEN UDP_Send.RecordTime := SCC_RecordTime; END_IF
IF NOT _w3 THEN UDP_Send.RecordTime := VCC_RecordTime; END_IF

END_PROGRAM

// IndraMotionMlc1/Application/Input_Signals
FUNCTION_BLOCK Input_Signals
VAR_INPUT
END_VAR
VAR_OUTPUT
	Pressure_p001: REAL;
	Pressure_p002: REAL;
	Pressure_p003: REAL;
	Pressure_p004: REAL;
	Pressure_p005: REAL;
	Pressure_p006: REAL;
	Pressure_p007: REAL;
	Pressure_p008: REAL;
	Pressure_p009: REAL;
	Pressure_p010: REAL;
	Pressure_p011: REAL;
	Temperature_T004: REAL;
	Temperature_T006: REAL;
	Temperature_T011: REAL;
	Position_s021: REAL; 
	Pressure_pP: REAL;
	Pressure_pR: REAL;
	Pressure_pA: REAL;
	Pressure_pA1: REAL;
	Pressure_pB: REAL; 
	Pressure_pC: REAL;
	Flow_QB: REAL; 
	PVG_Valve_Opening: REAL;
	PRV_Valve_Opening: REAL;
	// Accelerometer
	Acc_Y_act: REAL;
	Acc_Y: REAL;
END_VAR
VAR
	FIR_FIlter_0: FIR_FIlter;
	Low_Pass_Filter_1: Low_Pass_Filter;
	LP_Num: LREAL := 0.9516;
	LP_Den: LREAL := 0.9048;
	FIR: LREAL := 0.5;
	FIR_FIlter_1: FIR_FIlter;
	FIR_FIlter_2: FIR_FIlter;
	Acc_Y_0: REAL := 15016;
	T_LPF: LREAL := 0.05;
	K_LPF: LREAL := 1;
	T4_scaling: REAL := 300;
	T11_scaling: REAL := 300;
	T4_correction: REAL := 0;
	T11_correction: REAL := 0;
	Discrete_Lowpass_Filter0_0: Discrete_Lowpass_Filter0;
END_VAR
VAR // added by the converter: edge detectors and wires of the graphical bodies
    _w1, _w2, _w3, _w4, _w5, _w6, _w7, _w8, _w9, _w10, _w11, _w12, _w13, _w14, _w15, _w16, _w17, _w18, _w19, _w20, _w21, _w22, _w23, _w24, _w25 : INT;
END_VAR

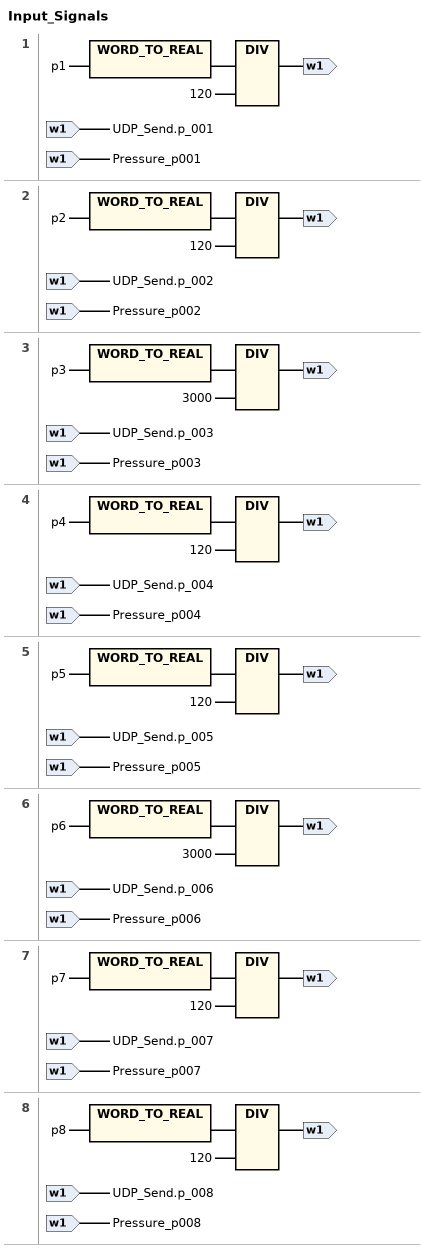
// NETWORK 1
_w1 := WORD_TO_REAL(p1) / 120;
UDP_Send.p_001 := _w1;
Pressure_p001 := _w1;

// NETWORK 2
_w2 := WORD_TO_REAL(p2) / 120;
UDP_Send.p_002 := _w2;
Pressure_p002 := _w2;

// NETWORK 3
_w3 := WORD_TO_REAL(p3) / 3000;
UDP_Send.p_003 := _w3;
Pressure_p003 := _w3;

// NETWORK 4
_w4 := WORD_TO_REAL(p4) / 120;
UDP_Send.p_004 := _w4;
Pressure_p004 := _w4;

// NETWORK 5
_w5 := WORD_TO_REAL(p5) / 120;
UDP_Send.p_005 := _w5;
Pressure_p005 := _w5;

// NETWORK 6
_w6 := WORD_TO_REAL(p6) / 3000;
UDP_Send.p_006 := _w6;
Pressure_p006 := _w6;

// NETWORK 7
_w7 := WORD_TO_REAL(p7) / 120;
UDP_Send.p_007 := _w7;
Pressure_p007 := _w7;

// NETWORK 8
_w8 := WORD_TO_REAL(p8) / 120;
UDP_Send.p_008 := _w8;
Pressure_p008 := _w8;

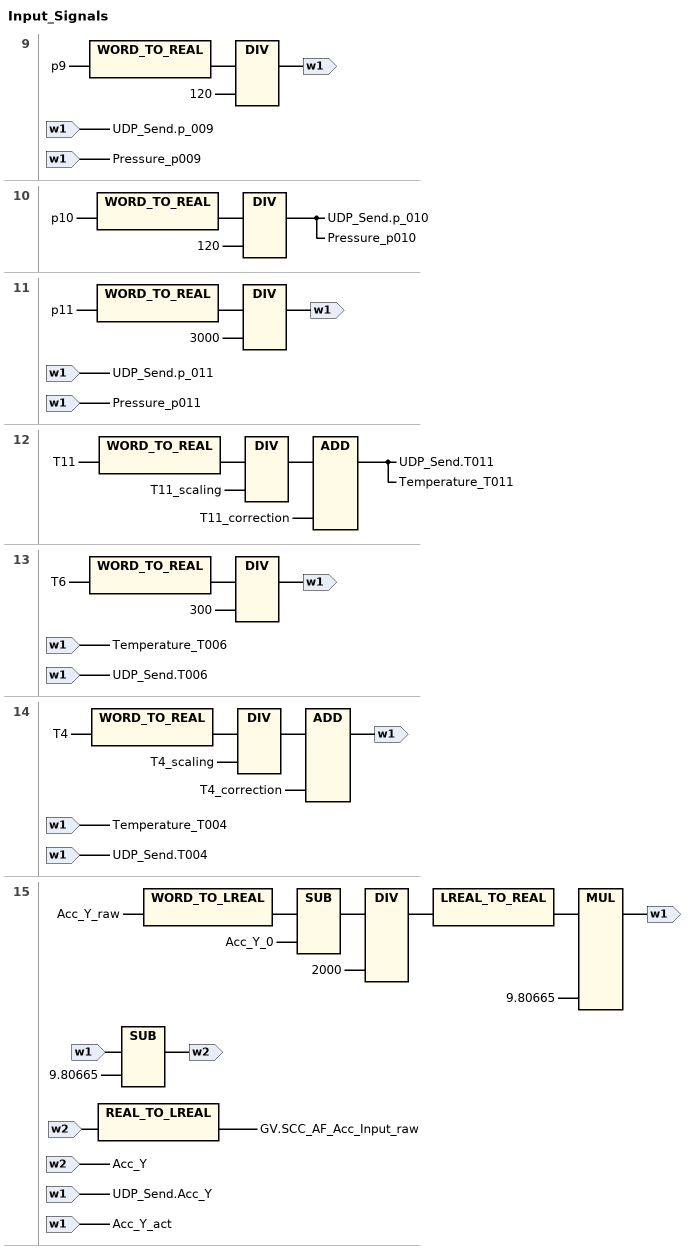
// NETWORK 9
_w9 := WORD_TO_REAL(p9) / 120;
UDP_Send.p_009 := _w9;
Pressure_p009 := _w9;

// NETWORK 10
_w10 := WORD_TO_REAL(p10) / 120;
UDP_Send.p_010 := _w10;
Pressure_p010 := _w10;

// NETWORK 11
_w11 := WORD_TO_REAL(p11) / 3000;
UDP_Send.p_011 := _w11;
Pressure_p011 := _w11;

// NETWORK 12
_w12 := WORD_TO_REAL(T11) / T11_scaling + T11_correction;
UDP_Send.T011 := _w12;
Temperature_T011 := _w12;

// NETWORK 13
_w13 := WORD_TO_REAL(T6) / 300;
Temperature_T006 := _w13;
UDP_Send.T006 := _w13;

// NETWORK 14
_w14 := WORD_TO_REAL(T4) / T4_scaling + T4_correction;
Temperature_T004 := _w14;
UDP_Send.T004 := _w14;

// NETWORK 15
_w15 := LREAL_TO_REAL((WORD_TO_LREAL(Acc_Y_raw) - Acc_Y_0) / 2000) * 9.80665;
_w16 := _w15 - 9.80665;
GV.SCC_AF_Acc_Input_raw := REAL_TO_LREAL(_w16);
Acc_Y := _w16;
UDP_Send.Acc_Y := _w15;
Acc_Y_act := _w15;

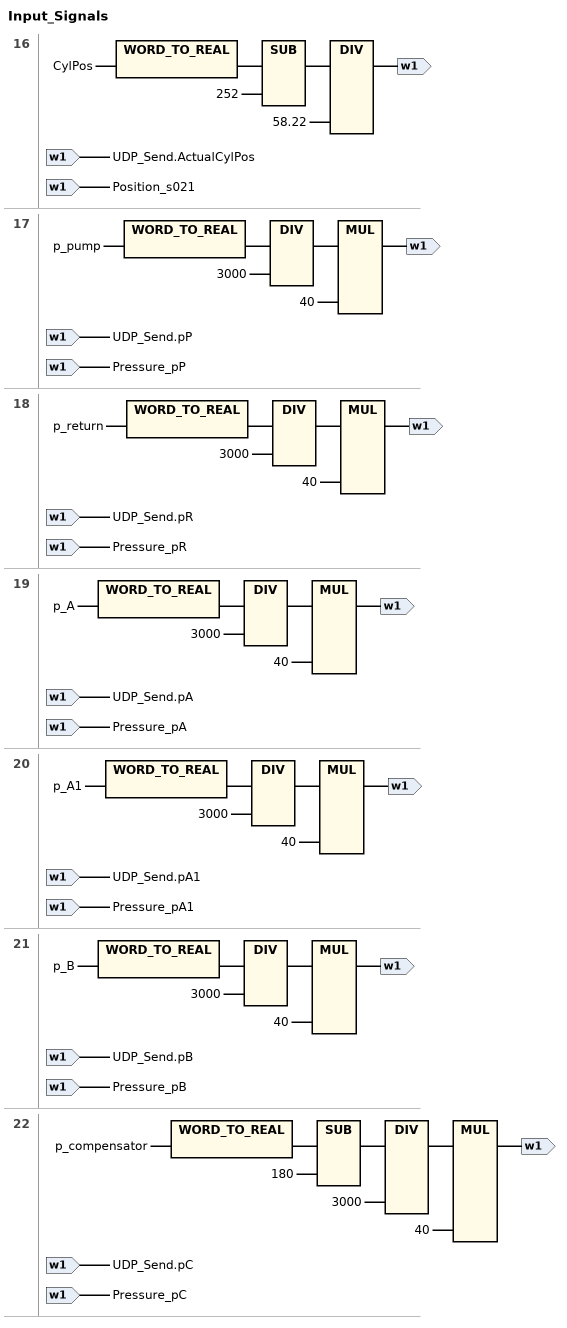
// NETWORK 16
_w17 := (WORD_TO_REAL(CylPos) - 252) / 58.22;
UDP_Send.ActualCylPos := _w17;
Position_s021 := _w17;

// NETWORK 17
_w18 := (WORD_TO_REAL(p_pump) / 3000) * 40;
UDP_Send.pP := _w18;
Pressure_pP := _w18;

// NETWORK 18
_w19 := (WORD_TO_REAL(p_return) / 3000) * 40;
UDP_Send.pR := _w19;
Pressure_pR := _w19;

// NETWORK 19
_w20 := (WORD_TO_REAL(p_A) / 3000) * 40;
UDP_Send.pA := _w20;
Pressure_pA := _w20;

// NETWORK 20
_w21 := (WORD_TO_REAL(p_A1) / 3000) * 40;
UDP_Send.pA1 := _w21;
Pressure_pA1 := _w21;

// NETWORK 21
_w22 := (WORD_TO_REAL(p_B) / 3000) * 40;
UDP_Send.pB := _w22;
Pressure_pB := _w22;

// NETWORK 22
_w23 := ((WORD_TO_REAL(p_compensator) - 180) / 3000) * 40;
UDP_Send.pC := _w23;
Pressure_pC := _w23;

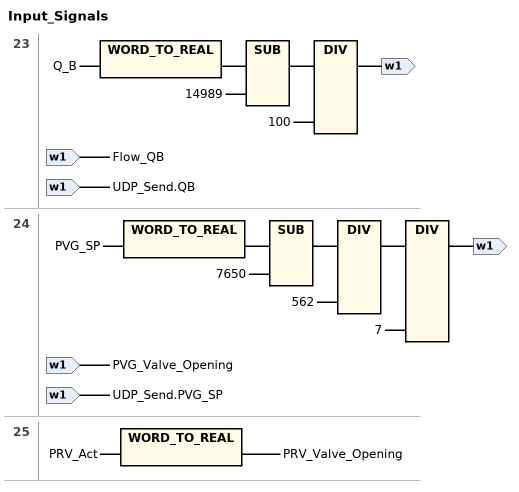
// NETWORK 23
_w24 := (WORD_TO_REAL(Q_B) - 14989) / 100;
Flow_QB := _w24;
UDP_Send.QB := _w24;

// NETWORK 24
_w25 := ((WORD_TO_REAL(PVG_SP) - 7650) / 562) / 7;
PVG_Valve_Opening := _w25;
UDP_Send.PVG_SP := _w25;

// NETWORK 25
PRV_Valve_Opening := WORD_TO_REAL(PRV_Act);

END_FUNCTION_BLOCK

// IndraMotionMlc1/Application/FIR_FIlter
FUNCTION_BLOCK FIR_FIlter
VAR_INPUT
	ssMethodType: SINT;
	In: LREAL;
END_VAR
VAR_OUTPUT
	Out: LREAL;
END_VAR
VAR
	j: DINT;
	DiscreteFIRFilter_states: LREAL;
END_VAR



CASE ssMethodType OF
    0: 
        (* InitializeConditions for DiscreteFir: '<S1>/Discrete FIR Filter' *)
        DiscreteFIRFilter_states := 0.0;
    1: 
        (* DiscreteFir: '<S1>/Discrete FIR Filter' *)
        (* Consume delay line and beginning of input samples *)
        Out := 0.0;
        j := 0;
        Out := (In * 0.5) + Out;
        j := 1;
        WHILE (j - 1) < 1 DO
            Out := (DiscreteFIRFilter_states * 0.5) + Out;
            j := j + 1;
        END_WHILE;
        (* Update delay line for next frame *)
        DiscreteFIRFilter_states := In;
        (* End of DiscreteFir: '<S1>/Discrete FIR Filter' *)
END_CASE;

END_FUNCTION_BLOCK

// IndraMotionMlc1/Application/Acc_Sensor
PROGRAM Acc_Sensor
VAR
	Acc_Y_0: LREAL := 15016;
	S_shape_Profile_0: S_shape_Profile;
END_VAR

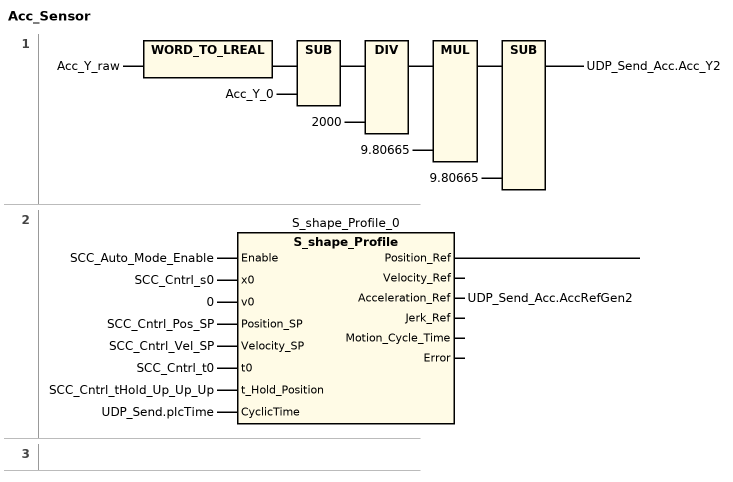
// NETWORK 1
UDP_Send_Acc.Acc_Y2 := ((WORD_TO_LREAL(Acc_Y_raw) - Acc_Y_0) / 2000) * 9.80665 - 9.80665;

// NETWORK 2
S_shape_Profile_0(
    Enable := SCC_Auto_Mode_Enable,
    x0 := SCC_Cntrl_s0,
    v0 := 0,
    Position_SP := SCC_Cntrl_Pos_SP,
    Velocity_SP := SCC_Cntrl_Vel_SP,
    t0 := SCC_Cntrl_t0,
    t_Hold_Position := SCC_Cntrl_tHold_Up_Up_Up,
    CyclicTime := UDP_Send.plcTime,
    Acceleration_Ref => UDP_Send_Acc.AccRefGen2); // S_shape_Profile

// NETWORK 3

END_PROGRAM

// IndraMotionMlc1/Application/CheckBounds
(*
General Header
----------------------------------------------------------------------------------------------
Short description      : Function to check access to array within valid bounds.
                         After inserting/removing this function, no online-change will be possible! A complete download will be necessary!
Version                : 14.1.0.0
Author                 : DC-IA/EAM3 (MD)
Date                   : 2015-01-12
Company                : Bosch Rexroth AG
Target                 : IndraLogic XLC/MLC
Functional description : This function will be called implicitly before the read/write access
                         to arrays takes places.
                         The index of the subsequent array accesses is checked for valid
                         limits.
                         In case of invalid access, an error is entered in the diagnostic
                         logbook and the application is stopped due to an access violation to
                         avoid machine damage.
                         In this case, check the callstack (menu Debug/Callstack) and modify
                         the faulty logic. 
Handling specials      : This function increases the cycle time of all IEC-tasks using array
                         accesses. 
                         The increase depends on the number of the read/write accesses to
                         arrays.
                         After inserting/removing this function, no online-change will be possible! 
                         A complete download will be necessary!
						 This is an exemplary implementation of the function. 
                         The implementation has to be adjusted to your application/machine.
						 Per default, the PLC-Task will generate an access violation which leads to
                         an application stop and a F5-error with error reaction respectively.
                         Please verify whether this default behaviour can damage your machine 
                         or lead to a complex recommissioning. 
                         In this case, adapt the error reaction to your application.
						 
                         If your application isn't too time-critical, you should leave this function 
						 while commissioning the machine and production in your application.  
                         If you remove this funciton, ensure that your code is faultless.
                         
                         Do not modify the declaration of this function! 
                         Do not change the attributes above the function header!
----------------------------------------------------------------------------------------------
*)
{attribute 'check_bounds'}
{attribute 'no_check'}
{attribute 'signature_flag' := '1073741824'}
FUNCTION CheckBounds : DINT
VAR_INPUT
	index, lower, upper: DINT;
END_VAR
VAR
	{attribute 'hide'}
	bByte: BYTE;
	ptNull: POINTER TO BYTE :=0;
	errstr: STRING;
	
END_VAR

